// TwinCAT 3 PLC project PLC
// ProgramVersion: 3.1.4023.0
// libraries:
//   Tc2_Standard, * (Beckhoff Automation GmbH)
//   Tc2_System, * (Beckhoff Automation GmbH)
//   Tc3_Module, * (Beckhoff Automation GmbH)
// project tree:
//   / PlcTask.TcTTO
//   POUs/ MAIN.TcPOU
//   DUTs/IO/PdoEntries/ Status_57491DF1.TcDUT, Status_D4FDECD4.TcDUT, Control_0B2F8B70.TcDUT, Status_B0753356.TcDUT, Status_F2CE6D91.TcDUT, Status_3A9E406C.TcDUT, Control_D500AB79.TcDUT, Status_D8D782C3.TcDUT, Control_6EF2C5D0.TcDUT, Status_8CBE219F.TcDUT, Status_B6795845.TcDUT, Control_5FD4673D.TcDUT, Status_1E008DB9.TcDUT, Status_3035BE2E.TcDUT, Control_F189B737.TcDUT, Control_C948E0F2.TcDUT, Status_6CCA259F.TcDUT, Status_72C27E80.TcDUT, Control_254441A5.TcDUT
//   DUTs/IO/PDOs/ InfoData_6F19DB2B.TcDUT, Channel_830843C1.TcDUT, WcState_9091E0EB.TcDUT, Latch_8E413295.TcDUT, WcState_B516A264.TcDUT, InfoData_A7436BC6.TcDUT, CNT_Input_Channel_FF10BD3C.TcDUT, DIG_Inputs_CAFF6004.TcDUT, DIG_Inputs_Device_1F4E72EB.TcDUT, CNT_Output_Channel_550BB6DF.TcDUT, InfoData_32EB74EA.TcDUT, Channel_42CA91F7.TcDUT, WcState_0B2B16F9.TcDUT, Diag_Channel_830843C1.TcDUT, InfoData_0A66F009.TcDUT, AI_Standard_Channel_A8DF64E3.TcDUT, RTD_RTDInputs_Channel_A8DF64E3.TcDUT, AI_Standard_Channel_4A394481.TcDUT, AO_Output_Channel_BA7EBB7C.TcDUT, AI_Inputs_Channel_A8DF64E3.TcDUT, ENC_Status_compact_F4F89583.TcDUT, ENC_Control_compact_E6DC9B25.TcDUT, ENC_Status_compact_7D3464F3.TcDUT, ENC_Control_compact_21E2D14D.TcDUT, COM_Inputs_6C2FC202.TcDUT, COM_Outputs_5D00B5E7.TcDUT, COM_TxPDO_Map_Inputs_Channel_C252EAC2.TcDUT, COM_RxPDO_Map_Outputs_Channel_B336F4EE.TcDUT, COM_TxPDO_Map_Inputs_Channel_6C2FC202.TcDUT, COM_RxPDO_Map_Outputs_Channel_5D00B5E7.TcDUT, ENC_Status_compact_4D066E1A.TcDUT, STM_Status_36ED096F.TcDUT, STM_Control_BA4CE352.TcDUT, STM_Velocity_A47A3F41.TcDUT, InfoData_6538CF5F.TcDUT, STM_Status_DE0D6B37.TcDUT, ENC_Status_compact_Channel_DC559AB0.TcDUT, DCM_Status_Channel_36ED096F.TcDUT, ENC_Control_compact_Channel_2E82BC43.TcDUT, DCM_Control_Channel_5A8B5016.TcDUT, DCM_Velocity_Channel_A47A3F41.TcDUT, InfoData_939F71B6.TcDUT, TACHO_Single_Shaft_Mode_Input_Channel_C331CA3E.TcDUT, DIG_Inputs_495F5DA4.TcDUT, PWM_Status_77939B11.TcDUT, DEV_Inputs_FBF180A4.TcDUT, TACHO_Output_Channel_600697D9.TcDUT, DIG_Outputs_0E284394.TcDUT, PWM_Control_63F162E4.TcDUT, InfoData_E68C61CD.TcDUT, InfoData_2A97D6CF.TcDUT, Inputs_25A0042B.TcDUT, Outputs_2397A10E.TcDUT
//   DUTs/IO/Boxes/ EK1100_1FC0878B.TcDUT, EK1122_1FC0878B.TcDUT, ER1008_78E8D3DD.TcDUT, ER1018_78E8D3DD.TcDUT, ER1098_78E8D3DD.TcDUT, ER1258_58F475DD.TcDUT, ER1518_CC442588.TcDUT, ER1809_32157CFD.TcDUT, ER1819_32157CFD.TcDUT, ER2008_E2806B95.TcDUT, ER2028_E2806B95.TcDUT, ER2038_3AE10DD7.TcDUT, ER2308_F6D9A8D1.TcDUT, ER2318_F6D9A8D1.TcDUT, ER2328_F6D9A8D1.TcDUT, ER2338_7699BCF6.TcDUT, ER2339_D8E9F29A.TcDUT, ER2339_4CF33DED.TcDUT, ER2349_4CF33DED.TcDUT, ER2624_7B64371E.TcDUT, ER2809_2B6483BD.TcDUT, ER3174_DCC78662.TcDUT, ER3184_DCC78662.TcDUT, ER3204_6CD7E119.TcDUT, ER3204_AB25C3AC.TcDUT, ER3314_E65CDB1C.TcDUT, ER4174_AB92710E.TcDUT, ER4374_A304750F.TcDUT, ER5101_87AC78CF.TcDUT, ER5151_7476E948.TcDUT, ER6001_40883D03.TcDUT, ER6002_7F53816A.TcDUT, ER6002_7BE6B617.TcDUT, ER7041_3210CF40.TcDUT, ER7041_3E4BEAEF.TcDUT, ER7342_2AE9C6B3.TcDUT, ER8309_A0C54F77.TcDUT
//   DUTs/IO/Devices/ SyncUnitTask_2D604ED5.TcDUT, SyncUnitTasks_6FEB8257.TcDUT, SyncUnits_99E584AF.TcDUT
//   DUTs/IO/Topology/ Beckhoff_ER1xxxEK1122_4914C526.TcDUT, Beckhoff_ER1xxx_A63E075A.TcDUT, Beckhoff_ER2xxxEK1122_73471FC4.TcDUT, Beckhoff_ER2xxx_CED8BB26.TcDUT, Beckhoff_ER3xxxEK1122_4F8E32D9.TcDUT, Beckhoff_ER3xxx_58A653D9.TcDUT, Beckhoff_ER4xxxEK1122_5C895096.TcDUT, Beckhoff_ER4xxx_797AEBB5.TcDUT, Beckhoff_ER5xxxEK1122_B89AF081.TcDUT, Beckhoff_ER5xxx_22A4CB20.TcDUT, Beckhoff_ER6xxxEK1122_BD5112F1.TcDUT, Beckhoff_ER6xxx_896D799E.TcDUT, Beckhoff_ER7xxxEK1122_0EBE6E72.TcDUT, Beckhoff_ER7xxx_FFC5AE47.TcDUT, Beckhoff_ER8xxxEK1122_CCFAC454.TcDUT, Beckhoff_ER8xxx_509945A9.TcDUT, EtherCAT_Master_ERxxxx_879C9A05.TcDUT
//   DUTs/IO/Base/ EtcSlaveBase_82538BE2.TcDUT, EtcSlaveBase_82538BE2.TcDUT, EtcSlaveBase_82538BE2.TcDUT, EtcSlaveTerminalBase_947E5A46.TcDUT, EtcSlaveBoxBase_77A0E4A7.TcDUT, EtcSlaveEndTerminalBase_866C7F0C.TcDUT, InputBase_8311D824.TcDUT, OutputBase_10CEE7DE.TcDUT, EtcMasterBase_62654B43.TcDUT
//   GVLs/ GVL_iXlinker.TcGVL
// real-time tasks:
//   TASK PlcTask: cycle T#10ms, priority 20, ADS port 350
// I/O:
//   DEVICE EtherCAT_Master_ERxxxx, AmsNetId 172.20.30.238.16.1
//     Beckhoff ER1xxx [EK1100 EtherCAT Coupler (2A E-Bus)]
//       Beckhoff ER1xxxEK1122 [EK1122 2 port EtherCAT junction]
//         Beckhoff ER1xxxsub EK1100 [EK1100 EtherCAT Coupler (2A E-Bus)]
//         A_0001(ER1008-0001-0016) [ER1008-0001 8 Ch. Dig. Input 24V, 3ms, M8]
//         A_0002(ER1008-0001-0018) [ER1008-0001 8 Ch. Dig. Input 24V, 3ms, M8]
//         A_0003(ER1008-0002-0018) [ER1008-0002 8 Ch. Dig. Input 24V, 3ms, M12]
//         A_0004(ER1008-0022-0017) [ER1008-0022 8 Ch. Dig. Input 24V, 3ms, M12]
//         A_0005(ER1018-0001-0018) [ER1018-0001 8 Ch. Dig. Input 24V, 10µs, M8]
//         A_0006(ER1018-0002-0018) [ER1018-0002 8 Ch. Dig. Input 24V, 10µs, M12]
//         A_0007(ER1098-0001-0017) [ER1098-0001 8 Ch. Dig. Input 24V, 10us, M8, negative]
//         A_0008(ER1258-0001-0019) [ER1258-0001 8 Ch. Dig. Input 24V, 10µs, DC Latch, M8]
//         A_0009(ER1258-0001-0020) [ER1258-0001 8 Ch. Dig. Input 24V, 10µs, DC Latch, M8]
//         A_0010(ER1258-0002-0019) [ER1258-0002 8 Ch. Dig. Input 24V, 10µs, DC Latch, M12]
//         A_0011(ER1258-0002-0020) [ER1258-0002 8 Ch. Dig. Input 24V, 10µs, DC Latch, M12]
//         A_0012(ER1518-0002-0018) [ER1518-0002 8 Ch.digital multi-function input]
//         A_0013(ER1518-0002-0019) [ER1518-0002 8 Ch.digital multi-function input]
//         A_0014(ER1809-0021-0017) [ER1809-0021 16 Ch. Dig. Input 24V, 3ms, M8]
//         A_0015(ER1809-0022-0018) [ER1809-0022 16 Ch. Dig. Input 24V, 3ms, M12]
//         A_0016(ER1819-0021-0017) [ER1819-0021 16 Ch. Dig. Input 24V, 10µs, M8]
//         A_0017(ER1819-0022-0017) [ER1819-0022 16 Ch. Dig. Input 24V, 10µs, M12]
//     Beckhoff ER2xxx [EK1100 EtherCAT Coupler (2A E-Bus)]
//       Beckhoff ER2xxxEK1122 [EK1122 2 port EtherCAT junction]
//         Beckhoff ER2xxxsub EK1100 [EK1100 EtherCAT Coupler (2A E-Bus)]
//         A_0001(ER2008-0001-0018) [ER2008-0001 8 Ch. Dig. Output 24V, 0,5A, M8]
//         A_0002(ER2008-0001-0019) [ER2008-0001 8 Ch. Dig. Output 24V, 0,5A, M8]
//         A_0003(ER2008-0002-0018) [ER2008-0002 8 Ch. Dig. Output 24V, 0,5A, M12]
//         A_0004(ER2008-0002-0019) [ER2008-0002 8 Ch. Dig. Output 24V, 0,5A, M12]
//         A_0005(ER2008-0022-0017) [ER2008-0022 8 Ch. Dig. Output 24V, 0,5A, M12]
//         A_0006(ER2008-0022-0018) [ER2008-0022 8 Ch. Dig. Output 24V, 0,5A, M12]
//         A_0007(ER2028-0001-0017) [ER2028-0001 8 Ch. Dig. Output 24V, 2A, M8]
//         A_0008(ER2028-0001-0018) [ER2028-0001 8 Ch. Dig. Output 24V, 2A, M8]
//         A_0009(ER2028-0002-0018) [ER2028-0002 8 Ch. Dig. Output 24V, 2A, M12]
//         A_0010(ER2028-0002-0019) [ER2028-0002 8 Ch. Dig. Output 24V, 2A, M12]
//         A_0011(ER2028-1032-0016) [ER2028-1032 8 Ch. Dig. Output 24V, 2,8A, M12]
//         A_0012(ER2038-0001-0017) [ER2038-0001 8 Ch. Dig. Output 24V, 2A, M8, Diagnostic]
//         A_0013(ER2038-0001-0018) [ER2038-0001 8 Ch. Dig. Output 24V, 2A, M8, Diagnostic]
//         A_0014(ER2038-0002-0017) [ER2038-0002 8 Ch. Dig. Output 24V, 2A, M12, Diagnostic]
//         A_0015(ER2038-0002-0018) [ER2038-0002 8 Ch. Dig. Output 24V, 2A, M12, Diagnostic]
//         A_0016(ER2308-0001-0018) [ER2308-0001 4 Ch. Dig. In, 3ms, 4 Ch. Dig. Out 24V, 0,5A, M8]
//         A_0017(ER2308-0001-0019) [ER2308-0001 4 Ch. Dig. In, 3ms, 4 Ch. Dig. Out 24V, 0,5A, M8]
//         A_0018(ER2308-0002-0018) [ER2308-0002 4 CH. Dig. In, 3ms, 4 Ch. Dig. Out 24V, 0,5A, M12]
//         A_0019(ER2308-0002-0019) [ER2308-0002 4 CH. Dig. In, 3ms, 4 Ch. Dig. Out 24V, 0,5A, M12]
//         A_0020(ER2318-0001-0018) [ER2318-0001 4 Ch. Dig. In, 10µs, 4 Ch. Dig. Out 24V, 0,5A, M8]
//         A_0021(ER2318-0001-0019) [ER2318-0001 4 Ch. Dig. In, 10µs, 4 Ch. Dig. Out 24V, 0,5A, M8]
//         A_0022(ER2318-0002-0018) [ER2318-0002 4 Ch. Dig. In, 10µs, 4 Ch. Dig. Out 24V, 0,5A, M12]
//         A_0023(ER2318-0002-0019) [ER2318-0002 4 Ch. Dig. In, 10µs, 4 Ch. Dig. Out 24V, 0,5A, M12]
//         A_0024(ER2328-0001-0017) [ER2328-0001 4 CH. Dig. In, 3ms, 4 Ch. Dig. Out 24V, 2A, M8]
//         A_0025(ER2328-0001-0018) [ER2328-0001 4 CH. Dig. In, 3ms, 4 Ch. Dig. Out 24V, 2A, M8]
//         A_0026(ER2328-0002-0018) [ER2328-0002 4 CH. Dig. In, 3ms, 4 Ch. Dig. Out 24V, 2A, M12]
//         A_0027(ER2328-0002-0019) [ER2328-0002 4 CH. Dig. In, 3ms, 4 Ch. Dig. Out 24V, 2A, M12]
//         A_0028(ER2338-0001-0022) [ER2338-0001 8 Ch. Dig. Input/Output 24V, 0,5A, M8]
//         A_0029(ER2338-0001-0023) [ER2338-0001 8 Ch. Dig. Input/Output 24V, 0,5A, M8]
//         A_0030(ER2338-0002-0022) [ER2338-0002 8 Ch. Dig. Input/Output 24V, 0,5A, M12]
//         A_0031(ER2338-0002-0023) [ER2338-0002 8 Ch. Dig. Input/Output 24V, 0,5A, M12]
//         A_0032(ER2338-1001-0017) [ER2338-1001 8 Ch. Dig. Input/Output 24V, 3ms, 0,5A, M8]
//         A_0033(ER2338-1001-0018) [ER2338-1001 8 Ch. Dig. Input/Output 24V, 3ms, 0,5A, M8]
//         A_0034(ER2338-1002-0017) [ER2338-1002 8 Ch. Dig. Input/Output 24V, 3ms, 0,5A, M12]
//         A_0035(ER2338-1002-0018) [ER2338-1002 8 Ch. Dig. Input/Output 24V, 3ms, 0,5A, M12]
//         A_0036(ER2339-0021-0018) [ER2339-0021 16 Ch. Dig. Input/Output 24V, 0,5A, M8]
//         A_0037(ER2339-0021-0019) [ER2339-0021 16 Ch. Dig. Input/Output 24V, 0,5A, M8]
//         A_0038(ER2339-0022-0018) [ER2339-0022 16 Ch. Dig. Input/Output 24V, 0,5A, M12]
//         A_0039(ER2339-0022-0019) [ER2339-0022 16 Ch. Dig. Input/Output 24V, 0,5A, M12]
//         A_0040(ER2349-0021-0017) [ER2349-0021 16 Ch. Dig. Input/Output 24V, 10µs, 0,5A, M8]
//         A_0041(ER2349-0021-0018) [ER2349-0021 16 Ch. Dig. Input/Output 24V, 10µs, 0,5A, M8]
//         A_0042(ER2349-0022-0017) [ER2349-0022 16 Ch. Dig. Input/Output 24V, 10µs, 0,5A, M12]
//         A_0043(ER2349-0022-0018) [ER2349-0022 16 Ch. Dig. Input/Output 24V, 10µs, 0,5A, M12]
//         A_0044(ER2624-0002-0018) [ER2624-0002 4Ch. Relay Output, NO (125V AC / 30V DC)]
//         A_0045(ER2624-0002-0019) [ER2624-0002 4Ch. Relay Output, NO (125V AC / 30V DC)]
//         A_0046(ER2809-0021-0017) [ER2809-0021 16 Ch. Dig. Output 24V, 0,5A, M8]
//         A_0047(ER2809-0021-0018) [ER2809-0021 16 Ch. Dig. Output 24V, 0,5A, M8]
//         A_0048(ER2809-0022-0016) [ER2809-0022 16 Ch. Dig. Output 24V, 0,5A, M12]
//         A_0049(ER2809-0022-0017) [ER2809-0022 16 Ch. Dig. Output 24V, 0,5A, M12]
//         A_0050(ER2809-0022-0018) [ER2809-0022 16 Ch. Dig. Output 24V, 0,5A, M12]
//     Beckhoff ER3xxx [EK1100 EtherCAT Coupler (2A E-Bus)]
//       Beckhoff ER3xxxEK1122 [EK1122 2 port EtherCAT junction]
//         Beckhoff ER3xxxsub EK1100 [EK1100 EtherCAT Coupler (2A E-Bus)]
//         A_0001(ER3174-0002-0016) [ER3174-0002 4Ch. Ana. Input +/-10V, 0-10V, 0/4-20mA configurable]
//         A_0002(ER3174-0002-0022) [ER3174-0002 4Ch. Ana. Input +/-10V, 0-10V, 0/4-20mA configurable]
//         A_0003(ER3174-0002-0023) [ER3174-0002 4Ch. Ana. Input +/-10V, 0-10V, 0/4-20mA configurable]
//         A_0004(ER3184-0002-0019) [ER3184-0002 4Ch. Ana. Input +/-10V, 0-10V, 0/4-20mA configurable, single ended]
//         A_0005(ER3184-0002-0020) [ER3184-0002 4Ch. Ana. Input +/-10V, 0-10V, 0/4-20mA configurable, single ended]
//         A_0006(ER3184-0002-0021) [ER3184-0002 4Ch. Ana. Input +/-10V, 0-10V, 0/4-20mA configurable, single ended]
//         A_0007(ER3184-1002-0020) [ER3184-1002 4Ch. Ana. Input +/-10V, 0-10V, 0/4-20mA configurable, single ended]
//         A_0008(ER3184-1002-0021) [ER3184-1002 4Ch. Ana. Input +/-10V, 0-10V, 0/4-20mA configurable, single ended]
//         A_0009(ER3204-0002-0016) [ER3204-0002 4Ch. Ana. Input PT100 (RTD)]
//         A_0010(ER3204-0002-0020) [ER3204-0002 4Ch. Ana. Input PT100 (RTD)]
//         A_0011(ER3204-0002-0021) [ER3204-0002 4Ch. Ana. Input PT100 (RTD)]
//         A_0012(ER3314-0002-0021) [ER3314-0002 4Ch. Ana. Input Thermocouple (TC)]
//     Beckhoff ER4xxx [EK1100 EtherCAT Coupler (2A E-Bus)]
//       Beckhoff ER4xxxEK1122 [EK1122 2 port EtherCAT junction]
//         Beckhoff ER4xxxsub EK1100 [EK1100 EtherCAT Coupler (2A E-Bus)]
//         A_0001(ER4174-0002-0016) [ER4174-0002 4Ch. Ana. Output +/-10V, 0-10V, 0/4-20mA configurable]
//         A_0002(ER4174-0002-0019) [ER4174-0002 4Ch. Ana. Output +/-10V, 0-10V, 0/4-20mA configurable]
//         A_0003(ER4374-0002-0018) [ER4374-0002 2Ch. Ana. Input +/-10V, 0-10V, 0/4-20mA configurable; 2Ch. Ana. Output +/-10V, 0-10V, 0/4-20mA configurable]
//         A_0004(ER4374-0002-0019) [ER4374-0002 2Ch. Ana. Input +/-10V, 0-10V, 0/4-20mA configurable; 2Ch. Ana. Output +/-10V, 0-10V, 0/4-20mA configurable]
//     Beckhoff ER5xxx [EK1100 EtherCAT Coupler (2A E-Bus)]
//       Beckhoff ER5xxxEK1122 [EK1122 2 port EtherCAT junction]
//         Beckhoff ER5xxxsub EK1100 [EK1100 EtherCAT Coupler (2A E-Bus)]
//         A_0001(ER5101-0002-0019) [ER5101-0002 1Ch. Inc. Encoder 5V, M12]
//         A_0002(ER5101-1002-0017) [ER5101-1002 1Ch. Inc. Encoder 5V, M12, 24V Sensor Supply]
//         A_0003(ER5151-0002-0018) [ER5151-0002 1Ch. Inc. Encoder 24V, M12, single ended]
//     Beckhoff ER6xxx [EK1100 EtherCAT Coupler (2A E-Bus)]
//       Beckhoff ER6xxxEK1122 [EK1122 2 port EtherCAT junction]
//         Beckhoff ER6xxxsub EK1100 [EK1100 EtherCAT Coupler (2A E-Bus)]
//         A_0001(ER6001-0002-0016) [ER6001-0002 Interface (RS232/422/485)]
//         A_0002(ER6001-0002-0021) [ER6001-0002 Interface (RS232/422/485)]
//         A_0003(ER6002-0002-0021) [ER6002-0002 Interface (RS232/422/485)]
//         A_0004(ER6002-0002-0022) [ER6002-0002 Interface (RS232/422/485)]
//         A_0005(ER6002-0002-0023) [ER6002-0002 Interface (RS232/422/485)]
//     Beckhoff ER7xxx [EK1100 EtherCAT Coupler (2A E-Bus)]
//       Beckhoff ER7xxxEK1122 [EK1122 2 port EtherCAT junction]
//         Beckhoff ER7xxxsub EK1100 [EK1100 EtherCAT Coupler (2A E-Bus)]
//         A_0001(ER7041-0002-0024) [ER7041-0002 1Ch. Stepper motor output stage (50V, 5A)]
//         A_0002(ER7041-0002-0025) [ER7041-0002 1Ch. Stepper motor output stage (50V, 5A)]
//         A_0003(ER7041-1002-0024) [ER7041-1002 1Ch. Stepper motor output stage (50V, 1.5A)]
//         A_0004(ER7041-1002-0025) [ER7041-1002 1Ch. Stepper motor output stage (50V, 1.5A)]
//         A_0005(ER7041-2002-0024) [ER7041-2002 1Ch. Stepper motor output stage (50V, 5A)]
//         A_0006(ER7041-2002-0025) [ER7041-2002 1Ch. Stepper motor output stage (50V, 5A)]
//         A_0007(ER7041-3002-0021) [ER7041-3002 1Ch. Stepper motor output stage (50V, 5A)]
//         A_0008(ER7041-3002-0022) [ER7041-3002 1Ch. Stepper motor output stage (50V, 5A)]
//         A_0009(ER7342-0002-0020) [ER7342-0002 2Ch. DC motor output stage (50V, 3.5A)]
//         A_0010(ER7342-0002-0021) [ER7342-0002 2Ch. DC motor output stage (50V, 3.5A)]
//         A_0011(ER7342-0002-0022) [ER7342-0002 2Ch. DC motor output stage (50V, 3.5A)]
//     Beckhoff ER8xxx [EK1100 EtherCAT Coupler (2A E-Bus)]
//       Beckhoff ER8xxxEK1122 [EK1122 2 port EtherCAT junction]
//         Beckhoff ER8xxxsub EK1100 [EK1100 EtherCAT Coupler (2A E-Bus)]
//         A_0001(ER8309-1022-0018) [ER8309-1022 2Ch. Ana. Input 4-20mA, 1Ch. Pulse Width Current Output (24V, 1.2A), 1 Ch Ana. Output, 2Ch Dig. Out 24V, 0.5A, 4Ch Dig. In. 24V, 4Ch Dig In/Out 24V, 0.5A, M12]
// variable links:
//   PLC/PLC Instance <-> EtherCAT Master ERxxxx/Beckhoff ER1xxx
//     PlcTask Inputs/GVL_iXlinker.EtherCAT_Master_ERxxxx.Beckhoff_ER1xxx.InfoData.State <-> InfoData/State
//   PLC/PLC Instance <-> EtherCAT Master ERxxxx/Beckhoff ER1xxx/Beckhoff ER1xxxEK1122
//     PlcTask Inputs/GVL_iXlinker.EtherCAT_Master_ERxxxx.Beckhoff_ER1xxx.Beckhoff_ER1xxxEK1122.InfoData.State <-> InfoData/State
//   PLC/PLC Instance <-> EtherCAT Master ERxxxx/Beckhoff ER1xxx/Beckhoff ER1xxxEK1122/Beckhoff ER1xxxsub EK1100
//     PlcTask Inputs/GVL_iXlinker.EtherCAT_Master_ERxxxx.Beckhoff_ER1xxx.Beckhoff_ER1xxxEK1122.Beckhoff_ER1xxxsub_EK1100.InfoData.State <-> InfoData/State
//   PLC/PLC Instance <-> EtherCAT Master ERxxxx/Beckhoff ER1xxx/Beckhoff ER1xxxEK1122/A_0001(ER1008-0001-0016)
//     PlcTask Inputs/GVL_iXlinker.EtherCAT_Master_ERxxxx.Beckhoff_ER1xxx.Beckhoff_ER1xxxEK1122.A_0001_ER1008_0001_0016.Channel_1.Input <-> Channel 1/Input
//     PlcTask Inputs/GVL_iXlinker.EtherCAT_Master_ERxxxx.Beckhoff_ER1xxx.Beckhoff_ER1xxxEK1122.A_0001_ER1008_0001_0016.Channel_2.Input <-> Channel 2/Input
//     PlcTask Inputs/GVL_iXlinker.EtherCAT_Master_ERxxxx.Beckhoff_ER1xxx.Beckhoff_ER1xxxEK1122.A_0001_ER1008_0001_0016.Channel_3.Input <-> Channel 3/Input
//     PlcTask Inputs/GVL_iXlinker.EtherCAT_Master_ERxxxx.Beckhoff_ER1xxx.Beckhoff_ER1xxxEK1122.A_0001_ER1008_0001_0016.Channel_4.Input <-> Channel 4/Input
//     PlcTask Inputs/GVL_iXlinker.EtherCAT_Master_ERxxxx.Beckhoff_ER1xxx.Beckhoff_ER1xxxEK1122.A_0001_ER1008_0001_0016.Channel_5.Input <-> Channel 5/Input
//     PlcTask Inputs/GVL_iXlinker.EtherCAT_Master_ERxxxx.Beckhoff_ER1xxx.Beckhoff_ER1xxxEK1122.A_0001_ER1008_0001_0016.Channel_6.Input <-> Channel 6/Input
//     PlcTask Inputs/GVL_iXlinker.EtherCAT_Master_ERxxxx.Beckhoff_ER1xxx.Beckhoff_ER1xxxEK1122.A_0001_ER1008_0001_0016.Channel_7.Input <-> Channel 7/Input
//     PlcTask Inputs/GVL_iXlinker.EtherCAT_Master_ERxxxx.Beckhoff_ER1xxx.Beckhoff_ER1xxxEK1122.A_0001_ER1008_0001_0016.Channel_8.Input <-> Channel 8/Input
//     PlcTask Inputs/GVL_iXlinker.EtherCAT_Master_ERxxxx.Beckhoff_ER1xxx.Beckhoff_ER1xxxEK1122.A_0001_ER1008_0001_0016.WcState.WcState <-> WcState/WcState
//     PlcTask Inputs/GVL_iXlinker.EtherCAT_Master_ERxxxx.Beckhoff_ER1xxx.Beckhoff_ER1xxxEK1122.A_0001_ER1008_0001_0016.WcState.InputToggle <-> WcState/InputToggle
//     PlcTask Inputs/GVL_iXlinker.EtherCAT_Master_ERxxxx.Beckhoff_ER1xxx.Beckhoff_ER1xxxEK1122.A_0001_ER1008_0001_0016.InfoData.State <-> InfoData/State
//   PLC/PLC Instance <-> EtherCAT Master ERxxxx/Beckhoff ER1xxx/Beckhoff ER1xxxEK1122/A_0002(ER1008-0001-0018)
//     PlcTask Inputs/GVL_iXlinker.EtherCAT_Master_ERxxxx.Beckhoff_ER1xxx.Beckhoff_ER1xxxEK1122.A_0002_ER1008_0001_0018.Channel_1.Input <-> Channel 1/Input
//     PlcTask Inputs/GVL_iXlinker.EtherCAT_Master_ERxxxx.Beckhoff_ER1xxx.Beckhoff_ER1xxxEK1122.A_0002_ER1008_0001_0018.Channel_2.Input <-> Channel 2/Input
//     PlcTask Inputs/GVL_iXlinker.EtherCAT_Master_ERxxxx.Beckhoff_ER1xxx.Beckhoff_ER1xxxEK1122.A_0002_ER1008_0001_0018.Channel_3.Input <-> Channel 3/Input
//     PlcTask Inputs/GVL_iXlinker.EtherCAT_Master_ERxxxx.Beckhoff_ER1xxx.Beckhoff_ER1xxxEK1122.A_0002_ER1008_0001_0018.Channel_4.Input <-> Channel 4/Input
//     PlcTask Inputs/GVL_iXlinker.EtherCAT_Master_ERxxxx.Beckhoff_ER1xxx.Beckhoff_ER1xxxEK1122.A_0002_ER1008_0001_0018.Channel_5.Input <-> Channel 5/Input
//     PlcTask Inputs/GVL_iXlinker.EtherCAT_Master_ERxxxx.Beckhoff_ER1xxx.Beckhoff_ER1xxxEK1122.A_0002_ER1008_0001_0018.Channel_6.Input <-> Channel 6/Input
//     PlcTask Inputs/GVL_iXlinker.EtherCAT_Master_ERxxxx.Beckhoff_ER1xxx.Beckhoff_ER1xxxEK1122.A_0002_ER1008_0001_0018.Channel_7.Input <-> Channel 7/Input
//     PlcTask Inputs/GVL_iXlinker.EtherCAT_Master_ERxxxx.Beckhoff_ER1xxx.Beckhoff_ER1xxxEK1122.A_0002_ER1008_0001_0018.Channel_8.Input <-> Channel 8/Input
//     PlcTask Inputs/GVL_iXlinker.EtherCAT_Master_ERxxxx.Beckhoff_ER1xxx.Beckhoff_ER1xxxEK1122.A_0002_ER1008_0001_0018.WcState.WcState <-> WcState/WcState
//     PlcTask Inputs/GVL_iXlinker.EtherCAT_Master_ERxxxx.Beckhoff_ER1xxx.Beckhoff_ER1xxxEK1122.A_0002_ER1008_0001_0018.WcState.InputToggle <-> WcState/InputToggle
//     PlcTask Inputs/GVL_iXlinker.EtherCAT_Master_ERxxxx.Beckhoff_ER1xxx.Beckhoff_ER1xxxEK1122.A_0002_ER1008_0001_0018.InfoData.State <-> InfoData/State
//   PLC/PLC Instance <-> EtherCAT Master ERxxxx/Beckhoff ER1xxx/Beckhoff ER1xxxEK1122/A_0003(ER1008-0002-0018)
//     PlcTask Inputs/GVL_iXlinker.EtherCAT_Master_ERxxxx.Beckhoff_ER1xxx.Beckhoff_ER1xxxEK1122.A_0003_ER1008_0002_0018.Channel_1.Input <-> Channel 1/Input
//     PlcTask Inputs/GVL_iXlinker.EtherCAT_Master_ERxxxx.Beckhoff_ER1xxx.Beckhoff_ER1xxxEK1122.A_0003_ER1008_0002_0018.Channel_2.Input <-> Channel 2/Input
//     PlcTask Inputs/GVL_iXlinker.EtherCAT_Master_ERxxxx.Beckhoff_ER1xxx.Beckhoff_ER1xxxEK1122.A_0003_ER1008_0002_0018.Channel_3.Input <-> Channel 3/Input
//     PlcTask Inputs/GVL_iXlinker.EtherCAT_Master_ERxxxx.Beckhoff_ER1xxx.Beckhoff_ER1xxxEK1122.A_0003_ER1008_0002_0018.Channel_4.Input <-> Channel 4/Input
//     PlcTask Inputs/GVL_iXlinker.EtherCAT_Master_ERxxxx.Beckhoff_ER1xxx.Beckhoff_ER1xxxEK1122.A_0003_ER1008_0002_0018.Channel_5.Input <-> Channel 5/Input
//     PlcTask Inputs/GVL_iXlinker.EtherCAT_Master_ERxxxx.Beckhoff_ER1xxx.Beckhoff_ER1xxxEK1122.A_0003_ER1008_0002_0018.Channel_6.Input <-> Channel 6/Input
//     PlcTask Inputs/GVL_iXlinker.EtherCAT_Master_ERxxxx.Beckhoff_ER1xxx.Beckhoff_ER1xxxEK1122.A_0003_ER1008_0002_0018.Channel_7.Input <-> Channel 7/Input
//     PlcTask Inputs/GVL_iXlinker.EtherCAT_Master_ERxxxx.Beckhoff_ER1xxx.Beckhoff_ER1xxxEK1122.A_0003_ER1008_0002_0018.Channel_8.Input <-> Channel 8/Input
//     PlcTask Inputs/GVL_iXlinker.EtherCAT_Master_ERxxxx.Beckhoff_ER1xxx.Beckhoff_ER1xxxEK1122.A_0003_ER1008_0002_0018.WcState.WcState <-> WcState/WcState
//     PlcTask Inputs/GVL_iXlinker.EtherCAT_Master_ERxxxx.Beckhoff_ER1xxx.Beckhoff_ER1xxxEK1122.A_0003_ER1008_0002_0018.WcState.InputToggle <-> WcState/InputToggle
//     PlcTask Inputs/GVL_iXlinker.EtherCAT_Master_ERxxxx.Beckhoff_ER1xxx.Beckhoff_ER1xxxEK1122.A_0003_ER1008_0002_0018.InfoData.State <-> InfoData/State
//   PLC/PLC Instance <-> EtherCAT Master ERxxxx/Beckhoff ER1xxx/Beckhoff ER1xxxEK1122/A_0004(ER1008-0022-0017)
//     PlcTask Inputs/GVL_iXlinker.EtherCAT_Master_ERxxxx.Beckhoff_ER1xxx.Beckhoff_ER1xxxEK1122.A_0004_ER1008_0022_0017.Channel_1.Input <-> Channel 1/Input
//     PlcTask Inputs/GVL_iXlinker.EtherCAT_Master_ERxxxx.Beckhoff_ER1xxx.Beckhoff_ER1xxxEK1122.A_0004_ER1008_0022_0017.Channel_2.Input <-> Channel 2/Input
//     PlcTask Inputs/GVL_iXlinker.EtherCAT_Master_ERxxxx.Beckhoff_ER1xxx.Beckhoff_ER1xxxEK1122.A_0004_ER1008_0022_0017.Channel_3.Input <-> Channel 3/Input
//     PlcTask Inputs/GVL_iXlinker.EtherCAT_Master_ERxxxx.Beckhoff_ER1xxx.Beckhoff_ER1xxxEK1122.A_0004_ER1008_0022_0017.Channel_4.Input <-> Channel 4/Input
//     PlcTask Inputs/GVL_iXlinker.EtherCAT_Master_ERxxxx.Beckhoff_ER1xxx.Beckhoff_ER1xxxEK1122.A_0004_ER1008_0022_0017.Channel_5.Input <-> Channel 5/Input
//     PlcTask Inputs/GVL_iXlinker.EtherCAT_Master_ERxxxx.Beckhoff_ER1xxx.Beckhoff_ER1xxxEK1122.A_0004_ER1008_0022_0017.Channel_6.Input <-> Channel 6/Input
//     PlcTask Inputs/GVL_iXlinker.EtherCAT_Master_ERxxxx.Beckhoff_ER1xxx.Beckhoff_ER1xxxEK1122.A_0004_ER1008_0022_0017.Channel_7.Input <-> Channel 7/Input
//     PlcTask Inputs/GVL_iXlinker.EtherCAT_Master_ERxxxx.Beckhoff_ER1xxx.Beckhoff_ER1xxxEK1122.A_0004_ER1008_0022_0017.Channel_8.Input <-> Channel 8/Input
//     PlcTask Inputs/GVL_iXlinker.EtherCAT_Master_ERxxxx.Beckhoff_ER1xxx.Beckhoff_ER1xxxEK1122.A_0004_ER1008_0022_0017.WcState.WcState <-> WcState/WcState
//     PlcTask Inputs/GVL_iXlinker.EtherCAT_Master_ERxxxx.Beckhoff_ER1xxx.Beckhoff_ER1xxxEK1122.A_0004_ER1008_0022_0017.WcState.InputToggle <-> WcState/InputToggle
//     PlcTask Inputs/GVL_iXlinker.EtherCAT_Master_ERxxxx.Beckhoff_ER1xxx.Beckhoff_ER1xxxEK1122.A_0004_ER1008_0022_0017.InfoData.State <-> InfoData/State
//   PLC/PLC Instance <-> EtherCAT Master ERxxxx/Beckhoff ER1xxx/Beckhoff ER1xxxEK1122/A_0005(ER1018-0001-0018)
//     PlcTask Inputs/GVL_iXlinker.EtherCAT_Master_ERxxxx.Beckhoff_ER1xxx.Beckhoff_ER1xxxEK1122.A_0005_ER1018_0001_0018.Channel_1.Input <-> Channel 1/Input
//     PlcTask Inputs/GVL_iXlinker.EtherCAT_Master_ERxxxx.Beckhoff_ER1xxx.Beckhoff_ER1xxxEK1122.A_0005_ER1018_0001_0018.Channel_2.Input <-> Channel 2/Input
//     PlcTask Inputs/GVL_iXlinker.EtherCAT_Master_ERxxxx.Beckhoff_ER1xxx.Beckhoff_ER1xxxEK1122.A_0005_ER1018_0001_0018.Channel_3.Input <-> Channel 3/Input
//     PlcTask Inputs/GVL_iXlinker.EtherCAT_Master_ERxxxx.Beckhoff_ER1xxx.Beckhoff_ER1xxxEK1122.A_0005_ER1018_0001_0018.Channel_4.Input <-> Channel 4/Input
//     PlcTask Inputs/GVL_iXlinker.EtherCAT_Master_ERxxxx.Beckhoff_ER1xxx.Beckhoff_ER1xxxEK1122.A_0005_ER1018_0001_0018.Channel_5.Input <-> Channel 5/Input
//     PlcTask Inputs/GVL_iXlinker.EtherCAT_Master_ERxxxx.Beckhoff_ER1xxx.Beckhoff_ER1xxxEK1122.A_0005_ER1018_0001_0018.Channel_6.Input <-> Channel 6/Input
//     PlcTask Inputs/GVL_iXlinker.EtherCAT_Master_ERxxxx.Beckhoff_ER1xxx.Beckhoff_ER1xxxEK1122.A_0005_ER1018_0001_0018.Channel_7.Input <-> Channel 7/Input
//     PlcTask Inputs/GVL_iXlinker.EtherCAT_Master_ERxxxx.Beckhoff_ER1xxx.Beckhoff_ER1xxxEK1122.A_0005_ER1018_0001_0018.Channel_8.Input <-> Channel 8/Input
//     PlcTask Inputs/GVL_iXlinker.EtherCAT_Master_ERxxxx.Beckhoff_ER1xxx.Beckhoff_ER1xxxEK1122.A_0005_ER1018_0001_0018.WcState.WcState <-> WcState/WcState
//     PlcTask Inputs/GVL_iXlinker.EtherCAT_Master_ERxxxx.Beckhoff_ER1xxx.Beckhoff_ER1xxxEK1122.A_0005_ER1018_0001_0018.WcState.InputToggle <-> WcState/InputToggle
//     PlcTask Inputs/GVL_iXlinker.EtherCAT_Master_ERxxxx.Beckhoff_ER1xxx.Beckhoff_ER1xxxEK1122.A_0005_ER1018_0001_0018.InfoData.State <-> InfoData/State
//   PLC/PLC Instance <-> EtherCAT Master ERxxxx/Beckhoff ER1xxx/Beckhoff ER1xxxEK1122/A_0006(ER1018-0002-0018)
//     PlcTask Inputs/GVL_iXlinker.EtherCAT_Master_ERxxxx.Beckhoff_ER1xxx.Beckhoff_ER1xxxEK1122.A_0006_ER1018_0002_0018.Channel_1.Input <-> Channel 1/Input
//     PlcTask Inputs/GVL_iXlinker.EtherCAT_Master_ERxxxx.Beckhoff_ER1xxx.Beckhoff_ER1xxxEK1122.A_0006_ER1018_0002_0018.Channel_2.Input <-> Channel 2/Input
//     PlcTask Inputs/GVL_iXlinker.EtherCAT_Master_ERxxxx.Beckhoff_ER1xxx.Beckhoff_ER1xxxEK1122.A_0006_ER1018_0002_0018.Channel_3.Input <-> Channel 3/Input
//     PlcTask Inputs/GVL_iXlinker.EtherCAT_Master_ERxxxx.Beckhoff_ER1xxx.Beckhoff_ER1xxxEK1122.A_0006_ER1018_0002_0018.Channel_4.Input <-> Channel 4/Input
//     PlcTask Inputs/GVL_iXlinker.EtherCAT_Master_ERxxxx.Beckhoff_ER1xxx.Beckhoff_ER1xxxEK1122.A_0006_ER1018_0002_0018.Channel_5.Input <-> Channel 5/Input
//     PlcTask Inputs/GVL_iXlinker.EtherCAT_Master_ERxxxx.Beckhoff_ER1xxx.Beckhoff_ER1xxxEK1122.A_0006_ER1018_0002_0018.Channel_6.Input <-> Channel 6/Input
//     PlcTask Inputs/GVL_iXlinker.EtherCAT_Master_ERxxxx.Beckhoff_ER1xxx.Beckhoff_ER1xxxEK1122.A_0006_ER1018_0002_0018.Channel_7.Input <-> Channel 7/Input
//     PlcTask Inputs/GVL_iXlinker.EtherCAT_Master_ERxxxx.Beckhoff_ER1xxx.Beckhoff_ER1xxxEK1122.A_0006_ER1018_0002_0018.Channel_8.Input <-> Channel 8/Input
//     PlcTask Inputs/GVL_iXlinker.EtherCAT_Master_ERxxxx.Beckhoff_ER1xxx.Beckhoff_ER1xxxEK1122.A_0006_ER1018_0002_0018.WcState.WcState <-> WcState/WcState
//     PlcTask Inputs/GVL_iXlinker.EtherCAT_Master_ERxxxx.Beckhoff_ER1xxx.Beckhoff_ER1xxxEK1122.A_0006_ER1018_0002_0018.WcState.InputToggle <-> WcState/InputToggle
//     PlcTask Inputs/GVL_iXlinker.EtherCAT_Master_ERxxxx.Beckhoff_ER1xxx.Beckhoff_ER1xxxEK1122.A_0006_ER1018_0002_0018.InfoData.State <-> InfoData/State
//   PLC/PLC Instance <-> EtherCAT Master ERxxxx/Beckhoff ER1xxx/Beckhoff ER1xxxEK1122/A_0007(ER1098-0001-0017)
//     PlcTask Inputs/GVL_iXlinker.EtherCAT_Master_ERxxxx.Beckhoff_ER1xxx.Beckhoff_ER1xxxEK1122.A_0007_ER1098_0001_0017.Channel_1.Input <-> Channel 1/Input
//     PlcTask Inputs/GVL_iXlinker.EtherCAT_Master_ERxxxx.Beckhoff_ER1xxx.Beckhoff_ER1xxxEK1122.A_0007_ER1098_0001_0017.Channel_2.Input <-> Channel 2/Input
//     PlcTask Inputs/GVL_iXlinker.EtherCAT_Master_ERxxxx.Beckhoff_ER1xxx.Beckhoff_ER1xxxEK1122.A_0007_ER1098_0001_0017.Channel_3.Input <-> Channel 3/Input
//     PlcTask Inputs/GVL_iXlinker.EtherCAT_Master_ERxxxx.Beckhoff_ER1xxx.Beckhoff_ER1xxxEK1122.A_0007_ER1098_0001_0017.Channel_4.Input <-> Channel 4/Input
//     PlcTask Inputs/GVL_iXlinker.EtherCAT_Master_ERxxxx.Beckhoff_ER1xxx.Beckhoff_ER1xxxEK1122.A_0007_ER1098_0001_0017.Channel_5.Input <-> Channel 5/Input
//     PlcTask Inputs/GVL_iXlinker.EtherCAT_Master_ERxxxx.Beckhoff_ER1xxx.Beckhoff_ER1xxxEK1122.A_0007_ER1098_0001_0017.Channel_6.Input <-> Channel 6/Input
//     PlcTask Inputs/GVL_iXlinker.EtherCAT_Master_ERxxxx.Beckhoff_ER1xxx.Beckhoff_ER1xxxEK1122.A_0007_ER1098_0001_0017.Channel_7.Input <-> Channel 7/Input
//     PlcTask Inputs/GVL_iXlinker.EtherCAT_Master_ERxxxx.Beckhoff_ER1xxx.Beckhoff_ER1xxxEK1122.A_0007_ER1098_0001_0017.Channel_8.Input <-> Channel 8/Input
//     PlcTask Inputs/GVL_iXlinker.EtherCAT_Master_ERxxxx.Beckhoff_ER1xxx.Beckhoff_ER1xxxEK1122.A_0007_ER1098_0001_0017.WcState.WcState <-> WcState/WcState
//     PlcTask Inputs/GVL_iXlinker.EtherCAT_Master_ERxxxx.Beckhoff_ER1xxx.Beckhoff_ER1xxxEK1122.A_0007_ER1098_0001_0017.WcState.InputToggle <-> WcState/InputToggle
//     PlcTask Inputs/GVL_iXlinker.EtherCAT_Master_ERxxxx.Beckhoff_ER1xxx.Beckhoff_ER1xxxEK1122.A_0007_ER1098_0001_0017.InfoData.State <-> InfoData/State
//   PLC/PLC Instance <-> EtherCAT Master ERxxxx/Beckhoff ER1xxx/Beckhoff ER1xxxEK1122/A_0008(ER1258-0001-0019)
//     PlcTask Inputs/GVL_iXlinker.EtherCAT_Master_ERxxxx.Beckhoff_ER1xxx.Beckhoff_ER1xxxEK1122.A_0008_ER1258_0001_0019.Channel_1.Input <-> Channel 1/Input
//     PlcTask Inputs/GVL_iXlinker.EtherCAT_Master_ERxxxx.Beckhoff_ER1xxx.Beckhoff_ER1xxxEK1122.A_0008_ER1258_0001_0019.Channel_2.Input <-> Channel 2/Input
//     PlcTask Inputs/GVL_iXlinker.EtherCAT_Master_ERxxxx.Beckhoff_ER1xxx.Beckhoff_ER1xxxEK1122.A_0008_ER1258_0001_0019.Channel_3.Input <-> Channel 3/Input
//     PlcTask Inputs/GVL_iXlinker.EtherCAT_Master_ERxxxx.Beckhoff_ER1xxx.Beckhoff_ER1xxxEK1122.A_0008_ER1258_0001_0019.Channel_4.Input <-> Channel 4/Input
//     PlcTask Inputs/GVL_iXlinker.EtherCAT_Master_ERxxxx.Beckhoff_ER1xxx.Beckhoff_ER1xxxEK1122.A_0008_ER1258_0001_0019.Channel_5.Input <-> Channel 5/Input
//     PlcTask Inputs/GVL_iXlinker.EtherCAT_Master_ERxxxx.Beckhoff_ER1xxx.Beckhoff_ER1xxxEK1122.A_0008_ER1258_0001_0019.Channel_6.Input <-> Channel 6/Input
//     PlcTask Inputs/GVL_iXlinker.EtherCAT_Master_ERxxxx.Beckhoff_ER1xxx.Beckhoff_ER1xxxEK1122.A_0008_ER1258_0001_0019.Channel_7.Input <-> Channel 7/Input
//     PlcTask Inputs/GVL_iXlinker.EtherCAT_Master_ERxxxx.Beckhoff_ER1xxx.Beckhoff_ER1xxxEK1122.A_0008_ER1258_0001_0019.Channel_8.Input <-> Channel 8/Input
//     PlcTask Inputs/GVL_iXlinker.EtherCAT_Master_ERxxxx.Beckhoff_ER1xxx.Beckhoff_ER1xxxEK1122.A_0008_ER1258_0001_0019.Latch.Status0 <-> Latch/Status0
//     PlcTask Inputs/GVL_iXlinker.EtherCAT_Master_ERxxxx.Beckhoff_ER1xxx.Beckhoff_ER1xxxEK1122.A_0008_ER1258_0001_0019.Latch.Status1 <-> Latch/Status1
//     PlcTask Inputs/GVL_iXlinker.EtherCAT_Master_ERxxxx.Beckhoff_ER1xxx.Beckhoff_ER1xxxEK1122.A_0008_ER1258_0001_0019.Latch.LatchPos0 <-> Latch/LatchPos0
//     PlcTask Inputs/GVL_iXlinker.EtherCAT_Master_ERxxxx.Beckhoff_ER1xxx.Beckhoff_ER1xxxEK1122.A_0008_ER1258_0001_0019.Latch.LatchPos1 <-> Latch/LatchPos1
//     PlcTask Inputs/GVL_iXlinker.EtherCAT_Master_ERxxxx.Beckhoff_ER1xxx.Beckhoff_ER1xxxEK1122.A_0008_ER1258_0001_0019.Latch.LatchNeg0 <-> Latch/LatchNeg0
//     PlcTask Inputs/GVL_iXlinker.EtherCAT_Master_ERxxxx.Beckhoff_ER1xxx.Beckhoff_ER1xxxEK1122.A_0008_ER1258_0001_0019.Latch.LatchNeg1 <-> Latch/LatchNeg1
//     PlcTask Inputs/GVL_iXlinker.EtherCAT_Master_ERxxxx.Beckhoff_ER1xxx.Beckhoff_ER1xxxEK1122.A_0008_ER1258_0001_0019.WcState.WcState0 <-> WcState/WcState0
//     PlcTask Inputs/GVL_iXlinker.EtherCAT_Master_ERxxxx.Beckhoff_ER1xxx.Beckhoff_ER1xxxEK1122.A_0008_ER1258_0001_0019.WcState.WcState1 <-> WcState/WcState1
//     PlcTask Inputs/GVL_iXlinker.EtherCAT_Master_ERxxxx.Beckhoff_ER1xxx.Beckhoff_ER1xxxEK1122.A_0008_ER1258_0001_0019.WcState.InputToggle0 <-> WcState/InputToggle0
//     PlcTask Inputs/GVL_iXlinker.EtherCAT_Master_ERxxxx.Beckhoff_ER1xxx.Beckhoff_ER1xxxEK1122.A_0008_ER1258_0001_0019.WcState.InputToggle1 <-> WcState/InputToggle1
//     PlcTask Inputs/GVL_iXlinker.EtherCAT_Master_ERxxxx.Beckhoff_ER1xxx.Beckhoff_ER1xxxEK1122.A_0008_ER1258_0001_0019.InfoData.DcOutputShift <-> InfoData/DcOutputShift
//     PlcTask Inputs/GVL_iXlinker.EtherCAT_Master_ERxxxx.Beckhoff_ER1xxx.Beckhoff_ER1xxxEK1122.A_0008_ER1258_0001_0019.InfoData.DcInputShift <-> InfoData/DcInputShift
//     PlcTask Inputs/GVL_iXlinker.EtherCAT_Master_ERxxxx.Beckhoff_ER1xxx.Beckhoff_ER1xxxEK1122.A_0008_ER1258_0001_0019.InfoData.State <-> InfoData/State
//   PLC/PLC Instance <-> EtherCAT Master ERxxxx/Beckhoff ER1xxx/Beckhoff ER1xxxEK1122/A_0009(ER1258-0001-0020)
//     PlcTask Inputs/GVL_iXlinker.EtherCAT_Master_ERxxxx.Beckhoff_ER1xxx.Beckhoff_ER1xxxEK1122.A_0009_ER1258_0001_0020.Channel_1.Input <-> Channel 1/Input
//     PlcTask Inputs/GVL_iXlinker.EtherCAT_Master_ERxxxx.Beckhoff_ER1xxx.Beckhoff_ER1xxxEK1122.A_0009_ER1258_0001_0020.Channel_2.Input <-> Channel 2/Input
//     PlcTask Inputs/GVL_iXlinker.EtherCAT_Master_ERxxxx.Beckhoff_ER1xxx.Beckhoff_ER1xxxEK1122.A_0009_ER1258_0001_0020.Channel_3.Input <-> Channel 3/Input
//     PlcTask Inputs/GVL_iXlinker.EtherCAT_Master_ERxxxx.Beckhoff_ER1xxx.Beckhoff_ER1xxxEK1122.A_0009_ER1258_0001_0020.Channel_4.Input <-> Channel 4/Input
//     PlcTask Inputs/GVL_iXlinker.EtherCAT_Master_ERxxxx.Beckhoff_ER1xxx.Beckhoff_ER1xxxEK1122.A_0009_ER1258_0001_0020.Channel_5.Input <-> Channel 5/Input
//     PlcTask Inputs/GVL_iXlinker.EtherCAT_Master_ERxxxx.Beckhoff_ER1xxx.Beckhoff_ER1xxxEK1122.A_0009_ER1258_0001_0020.Channel_6.Input <-> Channel 6/Input
//     PlcTask Inputs/GVL_iXlinker.EtherCAT_Master_ERxxxx.Beckhoff_ER1xxx.Beckhoff_ER1xxxEK1122.A_0009_ER1258_0001_0020.Channel_7.Input <-> Channel 7/Input
//     PlcTask Inputs/GVL_iXlinker.EtherCAT_Master_ERxxxx.Beckhoff_ER1xxx.Beckhoff_ER1xxxEK1122.A_0009_ER1258_0001_0020.Channel_8.Input <-> Channel 8/Input
//     PlcTask Inputs/GVL_iXlinker.EtherCAT_Master_ERxxxx.Beckhoff_ER1xxx.Beckhoff_ER1xxxEK1122.A_0009_ER1258_0001_0020.Latch.Status0 <-> Latch/Status0
//     PlcTask Inputs/GVL_iXlinker.EtherCAT_Master_ERxxxx.Beckhoff_ER1xxx.Beckhoff_ER1xxxEK1122.A_0009_ER1258_0001_0020.Latch.Status1 <-> Latch/Status1
//     PlcTask Inputs/GVL_iXlinker.EtherCAT_Master_ERxxxx.Beckhoff_ER1xxx.Beckhoff_ER1xxxEK1122.A_0009_ER1258_0001_0020.Latch.LatchPos0 <-> Latch/LatchPos0
//     PlcTask Inputs/GVL_iXlinker.EtherCAT_Master_ERxxxx.Beckhoff_ER1xxx.Beckhoff_ER1xxxEK1122.A_0009_ER1258_0001_0020.Latch.LatchPos1 <-> Latch/LatchPos1
//     PlcTask Inputs/GVL_iXlinker.EtherCAT_Master_ERxxxx.Beckhoff_ER1xxx.Beckhoff_ER1xxxEK1122.A_0009_ER1258_0001_0020.Latch.LatchNeg0 <-> Latch/LatchNeg0
//     PlcTask Inputs/GVL_iXlinker.EtherCAT_Master_ERxxxx.Beckhoff_ER1xxx.Beckhoff_ER1xxxEK1122.A_0009_ER1258_0001_0020.Latch.LatchNeg1 <-> Latch/LatchNeg1
//     PlcTask Inputs/GVL_iXlinker.EtherCAT_Master_ERxxxx.Beckhoff_ER1xxx.Beckhoff_ER1xxxEK1122.A_0009_ER1258_0001_0020.WcState.WcState0 <-> WcState/WcState0
//     PlcTask Inputs/GVL_iXlinker.EtherCAT_Master_ERxxxx.Beckhoff_ER1xxx.Beckhoff_ER1xxxEK1122.A_0009_ER1258_0001_0020.WcState.WcState1 <-> WcState/WcState1
//     PlcTask Inputs/GVL_iXlinker.EtherCAT_Master_ERxxxx.Beckhoff_ER1xxx.Beckhoff_ER1xxxEK1122.A_0009_ER1258_0001_0020.WcState.InputToggle0 <-> WcState/InputToggle0
//     PlcTask Inputs/GVL_iXlinker.EtherCAT_Master_ERxxxx.Beckhoff_ER1xxx.Beckhoff_ER1xxxEK1122.A_0009_ER1258_0001_0020.WcState.InputToggle1 <-> WcState/InputToggle1
//     PlcTask Inputs/GVL_iXlinker.EtherCAT_Master_ERxxxx.Beckhoff_ER1xxx.Beckhoff_ER1xxxEK1122.A_0009_ER1258_0001_0020.InfoData.DcOutputShift <-> InfoData/DcOutputShift
//     PlcTask Inputs/GVL_iXlinker.EtherCAT_Master_ERxxxx.Beckhoff_ER1xxx.Beckhoff_ER1xxxEK1122.A_0009_ER1258_0001_0020.InfoData.DcInputShift <-> InfoData/DcInputShift
//     PlcTask Inputs/GVL_iXlinker.EtherCAT_Master_ERxxxx.Beckhoff_ER1xxx.Beckhoff_ER1xxxEK1122.A_0009_ER1258_0001_0020.InfoData.State <-> InfoData/State
//   PLC/PLC Instance <-> EtherCAT Master ERxxxx/Beckhoff ER1xxx/Beckhoff ER1xxxEK1122/A_0010(ER1258-0002-0019)
//     PlcTask Inputs/GVL_iXlinker.EtherCAT_Master_ERxxxx.Beckhoff_ER1xxx.Beckhoff_ER1xxxEK1122.A_0010_ER1258_0002_0019.Channel_1.Input <-> Channel 1/Input
//     PlcTask Inputs/GVL_iXlinker.EtherCAT_Master_ERxxxx.Beckhoff_ER1xxx.Beckhoff_ER1xxxEK1122.A_0010_ER1258_0002_0019.Channel_2.Input <-> Channel 2/Input
//     PlcTask Inputs/GVL_iXlinker.EtherCAT_Master_ERxxxx.Beckhoff_ER1xxx.Beckhoff_ER1xxxEK1122.A_0010_ER1258_0002_0019.Channel_3.Input <-> Channel 3/Input
//     PlcTask Inputs/GVL_iXlinker.EtherCAT_Master_ERxxxx.Beckhoff_ER1xxx.Beckhoff_ER1xxxEK1122.A_0010_ER1258_0002_0019.Channel_4.Input <-> Channel 4/Input
//     PlcTask Inputs/GVL_iXlinker.EtherCAT_Master_ERxxxx.Beckhoff_ER1xxx.Beckhoff_ER1xxxEK1122.A_0010_ER1258_0002_0019.Channel_5.Input <-> Channel 5/Input
//     PlcTask Inputs/GVL_iXlinker.EtherCAT_Master_ERxxxx.Beckhoff_ER1xxx.Beckhoff_ER1xxxEK1122.A_0010_ER1258_0002_0019.Channel_6.Input <-> Channel 6/Input
//     PlcTask Inputs/GVL_iXlinker.EtherCAT_Master_ERxxxx.Beckhoff_ER1xxx.Beckhoff_ER1xxxEK1122.A_0010_ER1258_0002_0019.Channel_7.Input <-> Channel 7/Input
//     PlcTask Inputs/GVL_iXlinker.EtherCAT_Master_ERxxxx.Beckhoff_ER1xxx.Beckhoff_ER1xxxEK1122.A_0010_ER1258_0002_0019.Channel_8.Input <-> Channel 8/Input
//     PlcTask Inputs/GVL_iXlinker.EtherCAT_Master_ERxxxx.Beckhoff_ER1xxx.Beckhoff_ER1xxxEK1122.A_0010_ER1258_0002_0019.Latch.Status0 <-> Latch/Status0
//     PlcTask Inputs/GVL_iXlinker.EtherCAT_Master_ERxxxx.Beckhoff_ER1xxx.Beckhoff_ER1xxxEK1122.A_0010_ER1258_0002_0019.Latch.Status1 <-> Latch/Status1
//     PlcTask Inputs/GVL_iXlinker.EtherCAT_Master_ERxxxx.Beckhoff_ER1xxx.Beckhoff_ER1xxxEK1122.A_0010_ER1258_0002_0019.Latch.LatchPos0 <-> Latch/LatchPos0
//     PlcTask Inputs/GVL_iXlinker.EtherCAT_Master_ERxxxx.Beckhoff_ER1xxx.Beckhoff_ER1xxxEK1122.A_0010_ER1258_0002_0019.Latch.LatchPos1 <-> Latch/LatchPos1
//     PlcTask Inputs/GVL_iXlinker.EtherCAT_Master_ERxxxx.Beckhoff_ER1xxx.Beckhoff_ER1xxxEK1122.A_0010_ER1258_0002_0019.Latch.LatchNeg0 <-> Latch/LatchNeg0
//     PlcTask Inputs/GVL_iXlinker.EtherCAT_Master_ERxxxx.Beckhoff_ER1xxx.Beckhoff_ER1xxxEK1122.A_0010_ER1258_0002_0019.Latch.LatchNeg1 <-> Latch/LatchNeg1
//     PlcTask Inputs/GVL_iXlinker.EtherCAT_Master_ERxxxx.Beckhoff_ER1xxx.Beckhoff_ER1xxxEK1122.A_0010_ER1258_0002_0019.WcState.WcState0 <-> WcState/WcState0
//     PlcTask Inputs/GVL_iXlinker.EtherCAT_Master_ERxxxx.Beckhoff_ER1xxx.Beckhoff_ER1xxxEK1122.A_0010_ER1258_0002_0019.WcState.WcState1 <-> WcState/WcState1
//     PlcTask Inputs/GVL_iXlinker.EtherCAT_Master_ERxxxx.Beckhoff_ER1xxx.Beckhoff_ER1xxxEK1122.A_0010_ER1258_0002_0019.WcState.InputToggle0 <-> WcState/InputToggle0
//     PlcTask Inputs/GVL_iXlinker.EtherCAT_Master_ERxxxx.Beckhoff_ER1xxx.Beckhoff_ER1xxxEK1122.A_0010_ER1258_0002_0019.WcState.InputToggle1 <-> WcState/InputToggle1
//     PlcTask Inputs/GVL_iXlinker.EtherCAT_Master_ERxxxx.Beckhoff_ER1xxx.Beckhoff_ER1xxxEK1122.A_0010_ER1258_0002_0019.InfoData.DcOutputShift <-> InfoData/DcOutputShift
//     PlcTask Inputs/GVL_iXlinker.EtherCAT_Master_ERxxxx.Beckhoff_ER1xxx.Beckhoff_ER1xxxEK1122.A_0010_ER1258_0002_0019.InfoData.DcInputShift <-> InfoData/DcInputShift
//     PlcTask Inputs/GVL_iXlinker.EtherCAT_Master_ERxxxx.Beckhoff_ER1xxx.Beckhoff_ER1xxxEK1122.A_0010_ER1258_0002_0019.InfoData.State <-> InfoData/State
//   PLC/PLC Instance <-> EtherCAT Master ERxxxx/Beckhoff ER1xxx/Beckhoff ER1xxxEK1122/A_0011(ER1258-0002-0020)
//     PlcTask Inputs/GVL_iXlinker.EtherCAT_Master_ERxxxx.Beckhoff_ER1xxx.Beckhoff_ER1xxxEK1122.A_0011_ER1258_0002_0020.Channel_1.Input <-> Channel 1/Input
//     PlcTask Inputs/GVL_iXlinker.EtherCAT_Master_ERxxxx.Beckhoff_ER1xxx.Beckhoff_ER1xxxEK1122.A_0011_ER1258_0002_0020.Channel_2.Input <-> Channel 2/Input
//     PlcTask Inputs/GVL_iXlinker.EtherCAT_Master_ERxxxx.Beckhoff_ER1xxx.Beckhoff_ER1xxxEK1122.A_0011_ER1258_0002_0020.Channel_3.Input <-> Channel 3/Input
//     PlcTask Inputs/GVL_iXlinker.EtherCAT_Master_ERxxxx.Beckhoff_ER1xxx.Beckhoff_ER1xxxEK1122.A_0011_ER1258_0002_0020.Channel_4.Input <-> Channel 4/Input
//     PlcTask Inputs/GVL_iXlinker.EtherCAT_Master_ERxxxx.Beckhoff_ER1xxx.Beckhoff_ER1xxxEK1122.A_0011_ER1258_0002_0020.Channel_5.Input <-> Channel 5/Input
//     PlcTask Inputs/GVL_iXlinker.EtherCAT_Master_ERxxxx.Beckhoff_ER1xxx.Beckhoff_ER1xxxEK1122.A_0011_ER1258_0002_0020.Channel_6.Input <-> Channel 6/Input
//     PlcTask Inputs/GVL_iXlinker.EtherCAT_Master_ERxxxx.Beckhoff_ER1xxx.Beckhoff_ER1xxxEK1122.A_0011_ER1258_0002_0020.Channel_7.Input <-> Channel 7/Input
//     PlcTask Inputs/GVL_iXlinker.EtherCAT_Master_ERxxxx.Beckhoff_ER1xxx.Beckhoff_ER1xxxEK1122.A_0011_ER1258_0002_0020.Channel_8.Input <-> Channel 8/Input
//     PlcTask Inputs/GVL_iXlinker.EtherCAT_Master_ERxxxx.Beckhoff_ER1xxx.Beckhoff_ER1xxxEK1122.A_0011_ER1258_0002_0020.Latch.Status0 <-> Latch/Status0
//     PlcTask Inputs/GVL_iXlinker.EtherCAT_Master_ERxxxx.Beckhoff_ER1xxx.Beckhoff_ER1xxxEK1122.A_0011_ER1258_0002_0020.Latch.Status1 <-> Latch/Status1
//     PlcTask Inputs/GVL_iXlinker.EtherCAT_Master_ERxxxx.Beckhoff_ER1xxx.Beckhoff_ER1xxxEK1122.A_0011_ER1258_0002_0020.Latch.LatchPos0 <-> Latch/LatchPos0
//     PlcTask Inputs/GVL_iXlinker.EtherCAT_Master_ERxxxx.Beckhoff_ER1xxx.Beckhoff_ER1xxxEK1122.A_0011_ER1258_0002_0020.Latch.LatchPos1 <-> Latch/LatchPos1
//     PlcTask Inputs/GVL_iXlinker.EtherCAT_Master_ERxxxx.Beckhoff_ER1xxx.Beckhoff_ER1xxxEK1122.A_0011_ER1258_0002_0020.Latch.LatchNeg0 <-> Latch/LatchNeg0
//     PlcTask Inputs/GVL_iXlinker.EtherCAT_Master_ERxxxx.Beckhoff_ER1xxx.Beckhoff_ER1xxxEK1122.A_0011_ER1258_0002_0020.Latch.LatchNeg1 <-> Latch/LatchNeg1
//     PlcTask Inputs/GVL_iXlinker.EtherCAT_Master_ERxxxx.Beckhoff_ER1xxx.Beckhoff_ER1xxxEK1122.A_0011_ER1258_0002_0020.WcState.WcState0 <-> WcState/WcState0
//     PlcTask Inputs/GVL_iXlinker.EtherCAT_Master_ERxxxx.Beckhoff_ER1xxx.Beckhoff_ER1xxxEK1122.A_0011_ER1258_0002_0020.WcState.WcState1 <-> WcState/WcState1
//     PlcTask Inputs/GVL_iXlinker.EtherCAT_Master_ERxxxx.Beckhoff_ER1xxx.Beckhoff_ER1xxxEK1122.A_0011_ER1258_0002_0020.WcState.InputToggle0 <-> WcState/InputToggle0
//     PlcTask Inputs/GVL_iXlinker.EtherCAT_Master_ERxxxx.Beckhoff_ER1xxx.Beckhoff_ER1xxxEK1122.A_0011_ER1258_0002_0020.WcState.InputToggle1 <-> WcState/InputToggle1
//     PlcTask Inputs/GVL_iXlinker.EtherCAT_Master_ERxxxx.Beckhoff_ER1xxx.Beckhoff_ER1xxxEK1122.A_0011_ER1258_0002_0020.InfoData.DcOutputShift <-> InfoData/DcOutputShift
//     PlcTask Inputs/GVL_iXlinker.EtherCAT_Master_ERxxxx.Beckhoff_ER1xxx.Beckhoff_ER1xxxEK1122.A_0011_ER1258_0002_0020.InfoData.DcInputShift <-> InfoData/DcInputShift
//     PlcTask Inputs/GVL_iXlinker.EtherCAT_Master_ERxxxx.Beckhoff_ER1xxx.Beckhoff_ER1xxxEK1122.A_0011_ER1258_0002_0020.InfoData.State <-> InfoData/State
//   PLC/PLC Instance <-> EtherCAT Master ERxxxx/Beckhoff ER1xxx/Beckhoff ER1xxxEK1122/A_0012(ER1518-0002-0018)
//     PlcTask Inputs/GVL_iXlinker.EtherCAT_Master_ERxxxx.Beckhoff_ER1xxx.Beckhoff_ER1xxxEK1122.A_0012_ER1518_0002_0018.CNT_Input_Channel_1.Status/Set_counter_done <-> CNT Input Channel 1/Status/Set counter done
//     PlcTask Inputs/GVL_iXlinker.EtherCAT_Master_ERxxxx.Beckhoff_ER1xxx.Beckhoff_ER1xxxEK1122.A_0012_ER1518_0002_0018.CNT_Input_Channel_2.Status/Set_counter_done <-> CNT Input Channel 2/Status/Set counter done
//     PlcTask Inputs/GVL_iXlinker.EtherCAT_Master_ERxxxx.Beckhoff_ER1xxx.Beckhoff_ER1xxxEK1122.A_0012_ER1518_0002_0018.CNT_Input_Channel_1.Status/Counter_inhibited <-> CNT Input Channel 1/Status/Counter inhibited
//     PlcTask Inputs/GVL_iXlinker.EtherCAT_Master_ERxxxx.Beckhoff_ER1xxx.Beckhoff_ER1xxxEK1122.A_0012_ER1518_0002_0018.CNT_Input_Channel_2.Status/Counter_inhibited <-> CNT Input Channel 2/Status/Counter inhibited
//     PlcTask Inputs/GVL_iXlinker.EtherCAT_Master_ERxxxx.Beckhoff_ER1xxx.Beckhoff_ER1xxxEK1122.A_0012_ER1518_0002_0018.CNT_Input_Channel_1.Status/Status_of_input_UD <-> CNT Input Channel 1/Status/Status of input UD
//     PlcTask Inputs/GVL_iXlinker.EtherCAT_Master_ERxxxx.Beckhoff_ER1xxx.Beckhoff_ER1xxxEK1122.A_0012_ER1518_0002_0018.CNT_Input_Channel_2.Status/Status_of_input_UD <-> CNT Input Channel 2/Status/Status of input UD
//     PlcTask Inputs/GVL_iXlinker.EtherCAT_Master_ERxxxx.Beckhoff_ER1xxx.Beckhoff_ER1xxxEK1122.A_0012_ER1518_0002_0018.CNT_Input_Channel_1.Status/Status_of_input_clock <-> CNT Input Channel 1/Status/Status of input clock
//     PlcTask Inputs/GVL_iXlinker.EtherCAT_Master_ERxxxx.Beckhoff_ER1xxx.Beckhoff_ER1xxxEK1122.A_0012_ER1518_0002_0018.CNT_Input_Channel_2.Status/Status_of_input_clock <-> CNT Input Channel 2/Status/Status of input clock
//     PlcTask Inputs/GVL_iXlinker.EtherCAT_Master_ERxxxx.Beckhoff_ER1xxx.Beckhoff_ER1xxxEK1122.A_0012_ER1518_0002_0018.CNT_Input_Channel_1.Status/Sync_error <-> CNT Input Channel 1/Status/Sync error
//     PlcTask Inputs/GVL_iXlinker.EtherCAT_Master_ERxxxx.Beckhoff_ER1xxx.Beckhoff_ER1xxxEK1122.A_0012_ER1518_0002_0018.CNT_Input_Channel_2.Status/Sync_error <-> CNT Input Channel 2/Status/Sync error
//     PlcTask Inputs/GVL_iXlinker.EtherCAT_Master_ERxxxx.Beckhoff_ER1xxx.Beckhoff_ER1xxxEK1122.A_0012_ER1518_0002_0018.CNT_Input_Channel_1.Status/TxPDO_State <-> CNT Input Channel 1/Status/TxPDO State
//     PlcTask Inputs/GVL_iXlinker.EtherCAT_Master_ERxxxx.Beckhoff_ER1xxx.Beckhoff_ER1xxxEK1122.A_0012_ER1518_0002_0018.CNT_Input_Channel_2.Status/TxPDO_State <-> CNT Input Channel 2/Status/TxPDO State
//     PlcTask Inputs/GVL_iXlinker.EtherCAT_Master_ERxxxx.Beckhoff_ER1xxx.Beckhoff_ER1xxxEK1122.A_0012_ER1518_0002_0018.CNT_Input_Channel_1.Status/TxPDO_Toggle <-> CNT Input Channel 1/Status/TxPDO Toggle
//     PlcTask Inputs/GVL_iXlinker.EtherCAT_Master_ERxxxx.Beckhoff_ER1xxx.Beckhoff_ER1xxxEK1122.A_0012_ER1518_0002_0018.CNT_Input_Channel_2.Status/TxPDO_Toggle <-> CNT Input Channel 2/Status/TxPDO Toggle
//     PlcTask Inputs/GVL_iXlinker.EtherCAT_Master_ERxxxx.Beckhoff_ER1xxx.Beckhoff_ER1xxxEK1122.A_0012_ER1518_0002_0018.CNT_Input_Channel_1.Counter_value <-> CNT Input Channel 1/Counter value
//     PlcTask Inputs/GVL_iXlinker.EtherCAT_Master_ERxxxx.Beckhoff_ER1xxx.Beckhoff_ER1xxxEK1122.A_0012_ER1518_0002_0018.CNT_Input_Channel_2.Counter_value <-> CNT Input Channel 2/Counter value
//     PlcTask Inputs/GVL_iXlinker.EtherCAT_Master_ERxxxx.Beckhoff_ER1xxx.Beckhoff_ER1xxxEK1122.A_0012_ER1518_0002_0018.DIG_Inputs.Input[0] <-> DIG Inputs/Input 0
//     PlcTask Inputs/GVL_iXlinker.EtherCAT_Master_ERxxxx.Beckhoff_ER1xxx.Beckhoff_ER1xxxEK1122.A_0012_ER1518_0002_0018.DIG_Inputs.Input[1] <-> DIG Inputs/Input 1
//     PlcTask Inputs/GVL_iXlinker.EtherCAT_Master_ERxxxx.Beckhoff_ER1xxx.Beckhoff_ER1xxxEK1122.A_0012_ER1518_0002_0018.DIG_Inputs.Input[2] <-> DIG Inputs/Input 2
//     PlcTask Inputs/GVL_iXlinker.EtherCAT_Master_ERxxxx.Beckhoff_ER1xxx.Beckhoff_ER1xxxEK1122.A_0012_ER1518_0002_0018.DIG_Inputs.Input[3] <-> DIG Inputs/Input 3
//     PlcTask Inputs/GVL_iXlinker.EtherCAT_Master_ERxxxx.Beckhoff_ER1xxx.Beckhoff_ER1xxxEK1122.A_0012_ER1518_0002_0018.DIG_Inputs.Input[4] <-> DIG Inputs/Input 4
//     PlcTask Inputs/GVL_iXlinker.EtherCAT_Master_ERxxxx.Beckhoff_ER1xxx.Beckhoff_ER1xxxEK1122.A_0012_ER1518_0002_0018.DIG_Inputs.Input[5] <-> DIG Inputs/Input 5
//     PlcTask Inputs/GVL_iXlinker.EtherCAT_Master_ERxxxx.Beckhoff_ER1xxx.Beckhoff_ER1xxxEK1122.A_0012_ER1518_0002_0018.DIG_Inputs.Input[6] <-> DIG Inputs/Input 6
//     PlcTask Inputs/GVL_iXlinker.EtherCAT_Master_ERxxxx.Beckhoff_ER1xxx.Beckhoff_ER1xxxEK1122.A_0012_ER1518_0002_0018.DIG_Inputs.Input[7] <-> DIG Inputs/Input 7
//     PlcTask Inputs/GVL_iXlinker.EtherCAT_Master_ERxxxx.Beckhoff_ER1xxx.Beckhoff_ER1xxxEK1122.A_0012_ER1518_0002_0018.DIG_Inputs_Device.Status/Error_channel_1 <-> DIG Inputs Device/Status/Error channel 1
//     PlcTask Inputs/GVL_iXlinker.EtherCAT_Master_ERxxxx.Beckhoff_ER1xxx.Beckhoff_ER1xxxEK1122.A_0012_ER1518_0002_0018.DIG_Inputs_Device.Status/Error_channel_2 <-> DIG Inputs Device/Status/Error channel 2
//     PlcTask Inputs/GVL_iXlinker.EtherCAT_Master_ERxxxx.Beckhoff_ER1xxx.Beckhoff_ER1xxxEK1122.A_0012_ER1518_0002_0018.DIG_Inputs_Device.Status/Sync_error <-> DIG Inputs Device/Status/Sync error
//     PlcTask Inputs/GVL_iXlinker.EtherCAT_Master_ERxxxx.Beckhoff_ER1xxx.Beckhoff_ER1xxxEK1122.A_0012_ER1518_0002_0018.DIG_Inputs_Device.Status/TxPDO_State <-> DIG Inputs Device/Status/TxPDO State
//     PlcTask Inputs/GVL_iXlinker.EtherCAT_Master_ERxxxx.Beckhoff_ER1xxx.Beckhoff_ER1xxxEK1122.A_0012_ER1518_0002_0018.DIG_Inputs_Device.Status/TxPDO_Toggle <-> DIG Inputs Device/Status/TxPDO Toggle
//     PlcTask Outputs/GVL_iXlinker.EtherCAT_Master_ERxxxx.Beckhoff_ER1xxx.Beckhoff_ER1xxxEK1122.A_0012_ER1518_0002_0018.CNT_Output_Channel_1.Control/Set_counter <-> CNT Output Channel 1/Control/Set counter
//     PlcTask Outputs/GVL_iXlinker.EtherCAT_Master_ERxxxx.Beckhoff_ER1xxx.Beckhoff_ER1xxxEK1122.A_0012_ER1518_0002_0018.CNT_Output_Channel_2.Control/Set_counter <-> CNT Output Channel 2/Control/Set counter
//     PlcTask Outputs/GVL_iXlinker.EtherCAT_Master_ERxxxx.Beckhoff_ER1xxx.Beckhoff_ER1xxxEK1122.A_0012_ER1518_0002_0018.CNT_Output_Channel_1.Control/Inhibit_counter <-> CNT Output Channel 1/Control/Inhibit counter
//     PlcTask Outputs/GVL_iXlinker.EtherCAT_Master_ERxxxx.Beckhoff_ER1xxx.Beckhoff_ER1xxxEK1122.A_0012_ER1518_0002_0018.CNT_Output_Channel_2.Control/Inhibit_counter <-> CNT Output Channel 2/Control/Inhibit counter
//     PlcTask Outputs/GVL_iXlinker.EtherCAT_Master_ERxxxx.Beckhoff_ER1xxx.Beckhoff_ER1xxxEK1122.A_0012_ER1518_0002_0018.CNT_Output_Channel_1.Set_counter_value <-> CNT Output Channel 1/Set counter value
//     PlcTask Outputs/GVL_iXlinker.EtherCAT_Master_ERxxxx.Beckhoff_ER1xxx.Beckhoff_ER1xxxEK1122.A_0012_ER1518_0002_0018.CNT_Output_Channel_2.Set_counter_value <-> CNT Output Channel 2/Set counter value
//     PlcTask Inputs/GVL_iXlinker.EtherCAT_Master_ERxxxx.Beckhoff_ER1xxx.Beckhoff_ER1xxxEK1122.A_0012_ER1518_0002_0018.WcState.WcState <-> WcState/WcState
//     PlcTask Inputs/GVL_iXlinker.EtherCAT_Master_ERxxxx.Beckhoff_ER1xxx.Beckhoff_ER1xxxEK1122.A_0012_ER1518_0002_0018.WcState.InputToggle <-> WcState/InputToggle
//     PlcTask Inputs/GVL_iXlinker.EtherCAT_Master_ERxxxx.Beckhoff_ER1xxx.Beckhoff_ER1xxxEK1122.A_0012_ER1518_0002_0018.InfoData.AdsAddr <-> InfoData/AdsAddr
//     PlcTask Inputs/GVL_iXlinker.EtherCAT_Master_ERxxxx.Beckhoff_ER1xxx.Beckhoff_ER1xxxEK1122.A_0012_ER1518_0002_0018.InfoData.State <-> InfoData/State
//   PLC/PLC Instance <-> EtherCAT Master ERxxxx/Beckhoff ER1xxx/Beckhoff ER1xxxEK1122/A_0013(ER1518-0002-0019)
//     PlcTask Inputs/GVL_iXlinker.EtherCAT_Master_ERxxxx.Beckhoff_ER1xxx.Beckhoff_ER1xxxEK1122.A_0013_ER1518_0002_0019.CNT_Input_Channel_1.Status/Set_counter_done <-> CNT Input Channel 1/Status/Set counter done
//     PlcTask Inputs/GVL_iXlinker.EtherCAT_Master_ERxxxx.Beckhoff_ER1xxx.Beckhoff_ER1xxxEK1122.A_0013_ER1518_0002_0019.CNT_Input_Channel_2.Status/Set_counter_done <-> CNT Input Channel 2/Status/Set counter done
//     PlcTask Inputs/GVL_iXlinker.EtherCAT_Master_ERxxxx.Beckhoff_ER1xxx.Beckhoff_ER1xxxEK1122.A_0013_ER1518_0002_0019.CNT_Input_Channel_1.Status/Counter_inhibited <-> CNT Input Channel 1/Status/Counter inhibited
//     PlcTask Inputs/GVL_iXlinker.EtherCAT_Master_ERxxxx.Beckhoff_ER1xxx.Beckhoff_ER1xxxEK1122.A_0013_ER1518_0002_0019.CNT_Input_Channel_2.Status/Counter_inhibited <-> CNT Input Channel 2/Status/Counter inhibited
//     PlcTask Inputs/GVL_iXlinker.EtherCAT_Master_ERxxxx.Beckhoff_ER1xxx.Beckhoff_ER1xxxEK1122.A_0013_ER1518_0002_0019.CNT_Input_Channel_1.Status/Status_of_input_UD <-> CNT Input Channel 1/Status/Status of input UD
//     PlcTask Inputs/GVL_iXlinker.EtherCAT_Master_ERxxxx.Beckhoff_ER1xxx.Beckhoff_ER1xxxEK1122.A_0013_ER1518_0002_0019.CNT_Input_Channel_2.Status/Status_of_input_UD <-> CNT Input Channel 2/Status/Status of input UD
//     PlcTask Inputs/GVL_iXlinker.EtherCAT_Master_ERxxxx.Beckhoff_ER1xxx.Beckhoff_ER1xxxEK1122.A_0013_ER1518_0002_0019.CNT_Input_Channel_1.Status/Status_of_input_clock <-> CNT Input Channel 1/Status/Status of input clock
//     PlcTask Inputs/GVL_iXlinker.EtherCAT_Master_ERxxxx.Beckhoff_ER1xxx.Beckhoff_ER1xxxEK1122.A_0013_ER1518_0002_0019.CNT_Input_Channel_2.Status/Status_of_input_clock <-> CNT Input Channel 2/Status/Status of input clock
//     PlcTask Inputs/GVL_iXlinker.EtherCAT_Master_ERxxxx.Beckhoff_ER1xxx.Beckhoff_ER1xxxEK1122.A_0013_ER1518_0002_0019.CNT_Input_Channel_1.Status/Sync_error <-> CNT Input Channel 1/Status/Sync error
//     PlcTask Inputs/GVL_iXlinker.EtherCAT_Master_ERxxxx.Beckhoff_ER1xxx.Beckhoff_ER1xxxEK1122.A_0013_ER1518_0002_0019.CNT_Input_Channel_2.Status/Sync_error <-> CNT Input Channel 2/Status/Sync error
//     PlcTask Inputs/GVL_iXlinker.EtherCAT_Master_ERxxxx.Beckhoff_ER1xxx.Beckhoff_ER1xxxEK1122.A_0013_ER1518_0002_0019.CNT_Input_Channel_1.Status/TxPDO_State <-> CNT Input Channel 1/Status/TxPDO State
//     PlcTask Inputs/GVL_iXlinker.EtherCAT_Master_ERxxxx.Beckhoff_ER1xxx.Beckhoff_ER1xxxEK1122.A_0013_ER1518_0002_0019.CNT_Input_Channel_2.Status/TxPDO_State <-> CNT Input Channel 2/Status/TxPDO State
//     PlcTask Inputs/GVL_iXlinker.EtherCAT_Master_ERxxxx.Beckhoff_ER1xxx.Beckhoff_ER1xxxEK1122.A_0013_ER1518_0002_0019.CNT_Input_Channel_1.Status/TxPDO_Toggle <-> CNT Input Channel 1/Status/TxPDO Toggle
//     PlcTask Inputs/GVL_iXlinker.EtherCAT_Master_ERxxxx.Beckhoff_ER1xxx.Beckhoff_ER1xxxEK1122.A_0013_ER1518_0002_0019.CNT_Input_Channel_2.Status/TxPDO_Toggle <-> CNT Input Channel 2/Status/TxPDO Toggle
//     PlcTask Inputs/GVL_iXlinker.EtherCAT_Master_ERxxxx.Beckhoff_ER1xxx.Beckhoff_ER1xxxEK1122.A_0013_ER1518_0002_0019.CNT_Input_Channel_1.Counter_value <-> CNT Input Channel 1/Counter value
//     PlcTask Inputs/GVL_iXlinker.EtherCAT_Master_ERxxxx.Beckhoff_ER1xxx.Beckhoff_ER1xxxEK1122.A_0013_ER1518_0002_0019.CNT_Input_Channel_2.Counter_value <-> CNT Input Channel 2/Counter value
//     PlcTask Inputs/GVL_iXlinker.EtherCAT_Master_ERxxxx.Beckhoff_ER1xxx.Beckhoff_ER1xxxEK1122.A_0013_ER1518_0002_0019.DIG_Inputs.Input[0] <-> DIG Inputs/Input 0
//     PlcTask Inputs/GVL_iXlinker.EtherCAT_Master_ERxxxx.Beckhoff_ER1xxx.Beckhoff_ER1xxxEK1122.A_0013_ER1518_0002_0019.DIG_Inputs.Input[1] <-> DIG Inputs/Input 1
//     PlcTask Inputs/GVL_iXlinker.EtherCAT_Master_ERxxxx.Beckhoff_ER1xxx.Beckhoff_ER1xxxEK1122.A_0013_ER1518_0002_0019.DIG_Inputs.Input[2] <-> DIG Inputs/Input 2
//     PlcTask Inputs/GVL_iXlinker.EtherCAT_Master_ERxxxx.Beckhoff_ER1xxx.Beckhoff_ER1xxxEK1122.A_0013_ER1518_0002_0019.DIG_Inputs.Input[3] <-> DIG Inputs/Input 3
//     PlcTask Inputs/GVL_iXlinker.EtherCAT_Master_ERxxxx.Beckhoff_ER1xxx.Beckhoff_ER1xxxEK1122.A_0013_ER1518_0002_0019.DIG_Inputs.Input[4] <-> DIG Inputs/Input 4
//     PlcTask Inputs/GVL_iXlinker.EtherCAT_Master_ERxxxx.Beckhoff_ER1xxx.Beckhoff_ER1xxxEK1122.A_0013_ER1518_0002_0019.DIG_Inputs.Input[5] <-> DIG Inputs/Input 5
//     PlcTask Inputs/GVL_iXlinker.EtherCAT_Master_ERxxxx.Beckhoff_ER1xxx.Beckhoff_ER1xxxEK1122.A_0013_ER1518_0002_0019.DIG_Inputs.Input[6] <-> DIG Inputs/Input 6
//     PlcTask Inputs/GVL_iXlinker.EtherCAT_Master_ERxxxx.Beckhoff_ER1xxx.Beckhoff_ER1xxxEK1122.A_0013_ER1518_0002_0019.DIG_Inputs.Input[7] <-> DIG Inputs/Input 7
//     PlcTask Inputs/GVL_iXlinker.EtherCAT_Master_ERxxxx.Beckhoff_ER1xxx.Beckhoff_ER1xxxEK1122.A_0013_ER1518_0002_0019.DIG_Inputs_Device.Status/Error_channel_1 <-> DIG Inputs Device/Status/Error channel 1
//     PlcTask Inputs/GVL_iXlinker.EtherCAT_Master_ERxxxx.Beckhoff_ER1xxx.Beckhoff_ER1xxxEK1122.A_0013_ER1518_0002_0019.DIG_Inputs_Device.Status/Error_channel_2 <-> DIG Inputs Device/Status/Error channel 2
//     PlcTask Inputs/GVL_iXlinker.EtherCAT_Master_ERxxxx.Beckhoff_ER1xxx.Beckhoff_ER1xxxEK1122.A_0013_ER1518_0002_0019.DIG_Inputs_Device.Status/Sync_error <-> DIG Inputs Device/Status/Sync error
//     PlcTask Inputs/GVL_iXlinker.EtherCAT_Master_ERxxxx.Beckhoff_ER1xxx.Beckhoff_ER1xxxEK1122.A_0013_ER1518_0002_0019.DIG_Inputs_Device.Status/TxPDO_State <-> DIG Inputs Device/Status/TxPDO State
//     PlcTask Inputs/GVL_iXlinker.EtherCAT_Master_ERxxxx.Beckhoff_ER1xxx.Beckhoff_ER1xxxEK1122.A_0013_ER1518_0002_0019.DIG_Inputs_Device.Status/TxPDO_Toggle <-> DIG Inputs Device/Status/TxPDO Toggle
//     PlcTask Outputs/GVL_iXlinker.EtherCAT_Master_ERxxxx.Beckhoff_ER1xxx.Beckhoff_ER1xxxEK1122.A_0013_ER1518_0002_0019.CNT_Output_Channel_1.Control/Set_counter <-> CNT Output Channel 1/Control/Set counter
//     PlcTask Outputs/GVL_iXlinker.EtherCAT_Master_ERxxxx.Beckhoff_ER1xxx.Beckhoff_ER1xxxEK1122.A_0013_ER1518_0002_0019.CNT_Output_Channel_2.Control/Set_counter <-> CNT Output Channel 2/Control/Set counter
//     PlcTask Outputs/GVL_iXlinker.EtherCAT_Master_ERxxxx.Beckhoff_ER1xxx.Beckhoff_ER1xxxEK1122.A_0013_ER1518_0002_0019.CNT_Output_Channel_1.Control/Inhibit_counter <-> CNT Output Channel 1/Control/Inhibit counter
//     PlcTask Outputs/GVL_iXlinker.EtherCAT_Master_ERxxxx.Beckhoff_ER1xxx.Beckhoff_ER1xxxEK1122.A_0013_ER1518_0002_0019.CNT_Output_Channel_2.Control/Inhibit_counter <-> CNT Output Channel 2/Control/Inhibit counter
//     PlcTask Outputs/GVL_iXlinker.EtherCAT_Master_ERxxxx.Beckhoff_ER1xxx.Beckhoff_ER1xxxEK1122.A_0013_ER1518_0002_0019.CNT_Output_Channel_1.Set_counter_value <-> CNT Output Channel 1/Set counter value
//     PlcTask Outputs/GVL_iXlinker.EtherCAT_Master_ERxxxx.Beckhoff_ER1xxx.Beckhoff_ER1xxxEK1122.A_0013_ER1518_0002_0019.CNT_Output_Channel_2.Set_counter_value <-> CNT Output Channel 2/Set counter value
//     PlcTask Inputs/GVL_iXlinker.EtherCAT_Master_ERxxxx.Beckhoff_ER1xxx.Beckhoff_ER1xxxEK1122.A_0013_ER1518_0002_0019.WcState.WcState <-> WcState/WcState
//     PlcTask Inputs/GVL_iXlinker.EtherCAT_Master_ERxxxx.Beckhoff_ER1xxx.Beckhoff_ER1xxxEK1122.A_0013_ER1518_0002_0019.WcState.InputToggle <-> WcState/InputToggle
//     PlcTask Inputs/GVL_iXlinker.EtherCAT_Master_ERxxxx.Beckhoff_ER1xxx.Beckhoff_ER1xxxEK1122.A_0013_ER1518_0002_0019.InfoData.AdsAddr <-> InfoData/AdsAddr
//     PlcTask Inputs/GVL_iXlinker.EtherCAT_Master_ERxxxx.Beckhoff_ER1xxx.Beckhoff_ER1xxxEK1122.A_0013_ER1518_0002_0019.InfoData.State <-> InfoData/State
//   PLC/PLC Instance <-> EtherCAT Master ERxxxx/Beckhoff ER1xxx/Beckhoff ER1xxxEK1122/A_0014(ER1809-0021-0017)
//     PlcTask Inputs/GVL_iXlinker.EtherCAT_Master_ERxxxx.Beckhoff_ER1xxx.Beckhoff_ER1xxxEK1122.A_0014_ER1809_0021_0017.Channel_1.Input <-> Channel 1/Input
//     PlcTask Inputs/GVL_iXlinker.EtherCAT_Master_ERxxxx.Beckhoff_ER1xxx.Beckhoff_ER1xxxEK1122.A_0014_ER1809_0021_0017.Channel_2.Input <-> Channel 2/Input
//     PlcTask Inputs/GVL_iXlinker.EtherCAT_Master_ERxxxx.Beckhoff_ER1xxx.Beckhoff_ER1xxxEK1122.A_0014_ER1809_0021_0017.Channel_3.Input <-> Channel 3/Input
//     PlcTask Inputs/GVL_iXlinker.EtherCAT_Master_ERxxxx.Beckhoff_ER1xxx.Beckhoff_ER1xxxEK1122.A_0014_ER1809_0021_0017.Channel_4.Input <-> Channel 4/Input
//     PlcTask Inputs/GVL_iXlinker.EtherCAT_Master_ERxxxx.Beckhoff_ER1xxx.Beckhoff_ER1xxxEK1122.A_0014_ER1809_0021_0017.Channel_5.Input <-> Channel 5/Input
//     PlcTask Inputs/GVL_iXlinker.EtherCAT_Master_ERxxxx.Beckhoff_ER1xxx.Beckhoff_ER1xxxEK1122.A_0014_ER1809_0021_0017.Channel_6.Input <-> Channel 6/Input
//     PlcTask Inputs/GVL_iXlinker.EtherCAT_Master_ERxxxx.Beckhoff_ER1xxx.Beckhoff_ER1xxxEK1122.A_0014_ER1809_0021_0017.Channel_7.Input <-> Channel 7/Input
//     PlcTask Inputs/GVL_iXlinker.EtherCAT_Master_ERxxxx.Beckhoff_ER1xxx.Beckhoff_ER1xxxEK1122.A_0014_ER1809_0021_0017.Channel_8.Input <-> Channel 8/Input
//     PlcTask Inputs/GVL_iXlinker.EtherCAT_Master_ERxxxx.Beckhoff_ER1xxx.Beckhoff_ER1xxxEK1122.A_0014_ER1809_0021_0017.Channel_9.Input <-> Channel 9/Input
//     PlcTask Inputs/GVL_iXlinker.EtherCAT_Master_ERxxxx.Beckhoff_ER1xxx.Beckhoff_ER1xxxEK1122.A_0014_ER1809_0021_0017.Channel_10.Input <-> Channel 10/Input
//     PlcTask Inputs/GVL_iXlinker.EtherCAT_Master_ERxxxx.Beckhoff_ER1xxx.Beckhoff_ER1xxxEK1122.A_0014_ER1809_0021_0017.Channel_11.Input <-> Channel 11/Input
//     PlcTask Inputs/GVL_iXlinker.EtherCAT_Master_ERxxxx.Beckhoff_ER1xxx.Beckhoff_ER1xxxEK1122.A_0014_ER1809_0021_0017.Channel_12.Input <-> Channel 12/Input
//     PlcTask Inputs/GVL_iXlinker.EtherCAT_Master_ERxxxx.Beckhoff_ER1xxx.Beckhoff_ER1xxxEK1122.A_0014_ER1809_0021_0017.Channel_13.Input <-> Channel 13/Input
//     PlcTask Inputs/GVL_iXlinker.EtherCAT_Master_ERxxxx.Beckhoff_ER1xxx.Beckhoff_ER1xxxEK1122.A_0014_ER1809_0021_0017.Channel_14.Input <-> Channel 14/Input
//     PlcTask Inputs/GVL_iXlinker.EtherCAT_Master_ERxxxx.Beckhoff_ER1xxx.Beckhoff_ER1xxxEK1122.A_0014_ER1809_0021_0017.Channel_15.Input <-> Channel 15/Input
//     PlcTask Inputs/GVL_iXlinker.EtherCAT_Master_ERxxxx.Beckhoff_ER1xxx.Beckhoff_ER1xxxEK1122.A_0014_ER1809_0021_0017.Channel_16.Input <-> Channel 16/Input
//     PlcTask Inputs/GVL_iXlinker.EtherCAT_Master_ERxxxx.Beckhoff_ER1xxx.Beckhoff_ER1xxxEK1122.A_0014_ER1809_0021_0017.WcState.WcState <-> WcState/WcState
//     PlcTask Inputs/GVL_iXlinker.EtherCAT_Master_ERxxxx.Beckhoff_ER1xxx.Beckhoff_ER1xxxEK1122.A_0014_ER1809_0021_0017.WcState.InputToggle <-> WcState/InputToggle
//     PlcTask Inputs/GVL_iXlinker.EtherCAT_Master_ERxxxx.Beckhoff_ER1xxx.Beckhoff_ER1xxxEK1122.A_0014_ER1809_0021_0017.InfoData.State <-> InfoData/State
//   PLC/PLC Instance <-> EtherCAT Master ERxxxx/Beckhoff ER1xxx/Beckhoff ER1xxxEK1122/A_0015(ER1809-0022-0018)
//     PlcTask Inputs/GVL_iXlinker.EtherCAT_Master_ERxxxx.Beckhoff_ER1xxx.Beckhoff_ER1xxxEK1122.A_0015_ER1809_0022_0018.Channel_1.Input <-> Channel 1/Input
//     PlcTask Inputs/GVL_iXlinker.EtherCAT_Master_ERxxxx.Beckhoff_ER1xxx.Beckhoff_ER1xxxEK1122.A_0015_ER1809_0022_0018.Channel_2.Input <-> Channel 2/Input
//     PlcTask Inputs/GVL_iXlinker.EtherCAT_Master_ERxxxx.Beckhoff_ER1xxx.Beckhoff_ER1xxxEK1122.A_0015_ER1809_0022_0018.Channel_3.Input <-> Channel 3/Input
//     PlcTask Inputs/GVL_iXlinker.EtherCAT_Master_ERxxxx.Beckhoff_ER1xxx.Beckhoff_ER1xxxEK1122.A_0015_ER1809_0022_0018.Channel_4.Input <-> Channel 4/Input
//     PlcTask Inputs/GVL_iXlinker.EtherCAT_Master_ERxxxx.Beckhoff_ER1xxx.Beckhoff_ER1xxxEK1122.A_0015_ER1809_0022_0018.Channel_5.Input <-> Channel 5/Input
//     PlcTask Inputs/GVL_iXlinker.EtherCAT_Master_ERxxxx.Beckhoff_ER1xxx.Beckhoff_ER1xxxEK1122.A_0015_ER1809_0022_0018.Channel_6.Input <-> Channel 6/Input
//     PlcTask Inputs/GVL_iXlinker.EtherCAT_Master_ERxxxx.Beckhoff_ER1xxx.Beckhoff_ER1xxxEK1122.A_0015_ER1809_0022_0018.Channel_7.Input <-> Channel 7/Input
//     PlcTask Inputs/GVL_iXlinker.EtherCAT_Master_ERxxxx.Beckhoff_ER1xxx.Beckhoff_ER1xxxEK1122.A_0015_ER1809_0022_0018.Channel_8.Input <-> Channel 8/Input
//     PlcTask Inputs/GVL_iXlinker.EtherCAT_Master_ERxxxx.Beckhoff_ER1xxx.Beckhoff_ER1xxxEK1122.A_0015_ER1809_0022_0018.Channel_9.Input <-> Channel 9/Input
//     PlcTask Inputs/GVL_iXlinker.EtherCAT_Master_ERxxxx.Beckhoff_ER1xxx.Beckhoff_ER1xxxEK1122.A_0015_ER1809_0022_0018.Channel_10.Input <-> Channel 10/Input
//     PlcTask Inputs/GVL_iXlinker.EtherCAT_Master_ERxxxx.Beckhoff_ER1xxx.Beckhoff_ER1xxxEK1122.A_0015_ER1809_0022_0018.Channel_11.Input <-> Channel 11/Input
//     PlcTask Inputs/GVL_iXlinker.EtherCAT_Master_ERxxxx.Beckhoff_ER1xxx.Beckhoff_ER1xxxEK1122.A_0015_ER1809_0022_0018.Channel_12.Input <-> Channel 12/Input
//     PlcTask Inputs/GVL_iXlinker.EtherCAT_Master_ERxxxx.Beckhoff_ER1xxx.Beckhoff_ER1xxxEK1122.A_0015_ER1809_0022_0018.Channel_13.Input <-> Channel 13/Input
//     PlcTask Inputs/GVL_iXlinker.EtherCAT_Master_ERxxxx.Beckhoff_ER1xxx.Beckhoff_ER1xxxEK1122.A_0015_ER1809_0022_0018.Channel_14.Input <-> Channel 14/Input
//     PlcTask Inputs/GVL_iXlinker.EtherCAT_Master_ERxxxx.Beckhoff_ER1xxx.Beckhoff_ER1xxxEK1122.A_0015_ER1809_0022_0018.Channel_15.Input <-> Channel 15/Input
//     PlcTask Inputs/GVL_iXlinker.EtherCAT_Master_ERxxxx.Beckhoff_ER1xxx.Beckhoff_ER1xxxEK1122.A_0015_ER1809_0022_0018.Channel_16.Input <-> Channel 16/Input
//     PlcTask Inputs/GVL_iXlinker.EtherCAT_Master_ERxxxx.Beckhoff_ER1xxx.Beckhoff_ER1xxxEK1122.A_0015_ER1809_0022_0018.WcState.WcState <-> WcState/WcState
//     PlcTask Inputs/GVL_iXlinker.EtherCAT_Master_ERxxxx.Beckhoff_ER1xxx.Beckhoff_ER1xxxEK1122.A_0015_ER1809_0022_0018.WcState.InputToggle <-> WcState/InputToggle
//     PlcTask Inputs/GVL_iXlinker.EtherCAT_Master_ERxxxx.Beckhoff_ER1xxx.Beckhoff_ER1xxxEK1122.A_0015_ER1809_0022_0018.InfoData.State <-> InfoData/State
//   PLC/PLC Instance <-> EtherCAT Master ERxxxx/Beckhoff ER1xxx/Beckhoff ER1xxxEK1122/A_0016(ER1819-0021-0017)
//     PlcTask Inputs/GVL_iXlinker.EtherCAT_Master_ERxxxx.Beckhoff_ER1xxx.Beckhoff_ER1xxxEK1122.A_0016_ER1819_0021_0017.Channel_1.Input <-> Channel 1/Input
//     PlcTask Inputs/GVL_iXlinker.EtherCAT_Master_ERxxxx.Beckhoff_ER1xxx.Beckhoff_ER1xxxEK1122.A_0016_ER1819_0021_0017.Channel_2.Input <-> Channel 2/Input
//     PlcTask Inputs/GVL_iXlinker.EtherCAT_Master_ERxxxx.Beckhoff_ER1xxx.Beckhoff_ER1xxxEK1122.A_0016_ER1819_0021_0017.Channel_3.Input <-> Channel 3/Input
//     PlcTask Inputs/GVL_iXlinker.EtherCAT_Master_ERxxxx.Beckhoff_ER1xxx.Beckhoff_ER1xxxEK1122.A_0016_ER1819_0021_0017.Channel_4.Input <-> Channel 4/Input
//     PlcTask Inputs/GVL_iXlinker.EtherCAT_Master_ERxxxx.Beckhoff_ER1xxx.Beckhoff_ER1xxxEK1122.A_0016_ER1819_0021_0017.Channel_5.Input <-> Channel 5/Input
//     PlcTask Inputs/GVL_iXlinker.EtherCAT_Master_ERxxxx.Beckhoff_ER1xxx.Beckhoff_ER1xxxEK1122.A_0016_ER1819_0021_0017.Channel_6.Input <-> Channel 6/Input
//     PlcTask Inputs/GVL_iXlinker.EtherCAT_Master_ERxxxx.Beckhoff_ER1xxx.Beckhoff_ER1xxxEK1122.A_0016_ER1819_0021_0017.Channel_7.Input <-> Channel 7/Input
//     PlcTask Inputs/GVL_iXlinker.EtherCAT_Master_ERxxxx.Beckhoff_ER1xxx.Beckhoff_ER1xxxEK1122.A_0016_ER1819_0021_0017.Channel_8.Input <-> Channel 8/Input
//     PlcTask Inputs/GVL_iXlinker.EtherCAT_Master_ERxxxx.Beckhoff_ER1xxx.Beckhoff_ER1xxxEK1122.A_0016_ER1819_0021_0017.Channel_9.Input <-> Channel 9/Input
//     PlcTask Inputs/GVL_iXlinker.EtherCAT_Master_ERxxxx.Beckhoff_ER1xxx.Beckhoff_ER1xxxEK1122.A_0016_ER1819_0021_0017.Channel_10.Input <-> Channel 10/Input
//     PlcTask Inputs/GVL_iXlinker.EtherCAT_Master_ERxxxx.Beckhoff_ER1xxx.Beckhoff_ER1xxxEK1122.A_0016_ER1819_0021_0017.Channel_11.Input <-> Channel 11/Input
//     PlcTask Inputs/GVL_iXlinker.EtherCAT_Master_ERxxxx.Beckhoff_ER1xxx.Beckhoff_ER1xxxEK1122.A_0016_ER1819_0021_0017.Channel_12.Input <-> Channel 12/Input
//     PlcTask Inputs/GVL_iXlinker.EtherCAT_Master_ERxxxx.Beckhoff_ER1xxx.Beckhoff_ER1xxxEK1122.A_0016_ER1819_0021_0017.Channel_13.Input <-> Channel 13/Input
//     PlcTask Inputs/GVL_iXlinker.EtherCAT_Master_ERxxxx.Beckhoff_ER1xxx.Beckhoff_ER1xxxEK1122.A_0016_ER1819_0021_0017.Channel_14.Input <-> Channel 14/Input
//     PlcTask Inputs/GVL_iXlinker.EtherCAT_Master_ERxxxx.Beckhoff_ER1xxx.Beckhoff_ER1xxxEK1122.A_0016_ER1819_0021_0017.Channel_15.Input <-> Channel 15/Input
//     PlcTask Inputs/GVL_iXlinker.EtherCAT_Master_ERxxxx.Beckhoff_ER1xxx.Beckhoff_ER1xxxEK1122.A_0016_ER1819_0021_0017.Channel_16.Input <-> Channel 16/Input
//     PlcTask Inputs/GVL_iXlinker.EtherCAT_Master_ERxxxx.Beckhoff_ER1xxx.Beckhoff_ER1xxxEK1122.A_0016_ER1819_0021_0017.WcState.WcState <-> WcState/WcState
//     PlcTask Inputs/GVL_iXlinker.EtherCAT_Master_ERxxxx.Beckhoff_ER1xxx.Beckhoff_ER1xxxEK1122.A_0016_ER1819_0021_0017.WcState.InputToggle <-> WcState/InputToggle
//     PlcTask Inputs/GVL_iXlinker.EtherCAT_Master_ERxxxx.Beckhoff_ER1xxx.Beckhoff_ER1xxxEK1122.A_0016_ER1819_0021_0017.InfoData.State <-> InfoData/State
//   PLC/PLC Instance <-> EtherCAT Master ERxxxx/Beckhoff ER1xxx/Beckhoff ER1xxxEK1122/A_0017(ER1819-0022-0017)
//     PlcTask Inputs/GVL_iXlinker.EtherCAT_Master_ERxxxx.Beckhoff_ER1xxx.Beckhoff_ER1xxxEK1122.A_0017_ER1819_0022_0017.Channel_1.Input <-> Channel 1/Input
//     PlcTask Inputs/GVL_iXlinker.EtherCAT_Master_ERxxxx.Beckhoff_ER1xxx.Beckhoff_ER1xxxEK1122.A_0017_ER1819_0022_0017.Channel_2.Input <-> Channel 2/Input
//     PlcTask Inputs/GVL_iXlinker.EtherCAT_Master_ERxxxx.Beckhoff_ER1xxx.Beckhoff_ER1xxxEK1122.A_0017_ER1819_0022_0017.Channel_3.Input <-> Channel 3/Input
//     PlcTask Inputs/GVL_iXlinker.EtherCAT_Master_ERxxxx.Beckhoff_ER1xxx.Beckhoff_ER1xxxEK1122.A_0017_ER1819_0022_0017.Channel_4.Input <-> Channel 4/Input
//     PlcTask Inputs/GVL_iXlinker.EtherCAT_Master_ERxxxx.Beckhoff_ER1xxx.Beckhoff_ER1xxxEK1122.A_0017_ER1819_0022_0017.Channel_5.Input <-> Channel 5/Input
//     PlcTask Inputs/GVL_iXlinker.EtherCAT_Master_ERxxxx.Beckhoff_ER1xxx.Beckhoff_ER1xxxEK1122.A_0017_ER1819_0022_0017.Channel_6.Input <-> Channel 6/Input
//     PlcTask Inputs/GVL_iXlinker.EtherCAT_Master_ERxxxx.Beckhoff_ER1xxx.Beckhoff_ER1xxxEK1122.A_0017_ER1819_0022_0017.Channel_7.Input <-> Channel 7/Input
//     PlcTask Inputs/GVL_iXlinker.EtherCAT_Master_ERxxxx.Beckhoff_ER1xxx.Beckhoff_ER1xxxEK1122.A_0017_ER1819_0022_0017.Channel_8.Input <-> Channel 8/Input
//     PlcTask Inputs/GVL_iXlinker.EtherCAT_Master_ERxxxx.Beckhoff_ER1xxx.Beckhoff_ER1xxxEK1122.A_0017_ER1819_0022_0017.Channel_9.Input <-> Channel 9/Input
//     PlcTask Inputs/GVL_iXlinker.EtherCAT_Master_ERxxxx.Beckhoff_ER1xxx.Beckhoff_ER1xxxEK1122.A_0017_ER1819_0022_0017.Channel_10.Input <-> Channel 10/Input
//     PlcTask Inputs/GVL_iXlinker.EtherCAT_Master_ERxxxx.Beckhoff_ER1xxx.Beckhoff_ER1xxxEK1122.A_0017_ER1819_0022_0017.Channel_11.Input <-> Channel 11/Input
//     PlcTask Inputs/GVL_iXlinker.EtherCAT_Master_ERxxxx.Beckhoff_ER1xxx.Beckhoff_ER1xxxEK1122.A_0017_ER1819_0022_0017.Channel_12.Input <-> Channel 12/Input
//     PlcTask Inputs/GVL_iXlinker.EtherCAT_Master_ERxxxx.Beckhoff_ER1xxx.Beckhoff_ER1xxxEK1122.A_0017_ER1819_0022_0017.Channel_13.Input <-> Channel 13/Input
//     PlcTask Inputs/GVL_iXlinker.EtherCAT_Master_ERxxxx.Beckhoff_ER1xxx.Beckhoff_ER1xxxEK1122.A_0017_ER1819_0022_0017.Channel_14.Input <-> Channel 14/Input
//     PlcTask Inputs/GVL_iXlinker.EtherCAT_Master_ERxxxx.Beckhoff_ER1xxx.Beckhoff_ER1xxxEK1122.A_0017_ER1819_0022_0017.Channel_15.Input <-> Channel 15/Input
//     PlcTask Inputs/GVL_iXlinker.EtherCAT_Master_ERxxxx.Beckhoff_ER1xxx.Beckhoff_ER1xxxEK1122.A_0017_ER1819_0022_0017.Channel_16.Input <-> Channel 16/Input
//     PlcTask Inputs/GVL_iXlinker.EtherCAT_Master_ERxxxx.Beckhoff_ER1xxx.Beckhoff_ER1xxxEK1122.A_0017_ER1819_0022_0017.WcState.WcState <-> WcState/WcState
//     PlcTask Inputs/GVL_iXlinker.EtherCAT_Master_ERxxxx.Beckhoff_ER1xxx.Beckhoff_ER1xxxEK1122.A_0017_ER1819_0022_0017.WcState.InputToggle <-> WcState/InputToggle
//     PlcTask Inputs/GVL_iXlinker.EtherCAT_Master_ERxxxx.Beckhoff_ER1xxx.Beckhoff_ER1xxxEK1122.A_0017_ER1819_0022_0017.InfoData.State <-> InfoData/State
//   PLC/PLC Instance <-> EtherCAT Master ERxxxx/Beckhoff ER2xxx
//     PlcTask Inputs/GVL_iXlinker.EtherCAT_Master_ERxxxx.Beckhoff_ER2xxx.InfoData.State <-> InfoData/State
//   PLC/PLC Instance <-> EtherCAT Master ERxxxx/Beckhoff ER2xxx/Beckhoff ER2xxxEK1122
//     PlcTask Inputs/GVL_iXlinker.EtherCAT_Master_ERxxxx.Beckhoff_ER2xxx.Beckhoff_ER2xxxEK1122.InfoData.State <-> InfoData/State
//   PLC/PLC Instance <-> EtherCAT Master ERxxxx/Beckhoff ER2xxx/Beckhoff ER2xxxEK1122/Beckhoff ER2xxxsub EK1100
//     PlcTask Inputs/GVL_iXlinker.EtherCAT_Master_ERxxxx.Beckhoff_ER2xxx.Beckhoff_ER2xxxEK1122.Beckhoff_ER2xxxsub_EK1100.InfoData.State <-> InfoData/State
//   PLC/PLC Instance <-> EtherCAT Master ERxxxx/Beckhoff ER2xxx/Beckhoff ER2xxxEK1122/A_0001(ER2008-0001-0018)
//     PlcTask Outputs/GVL_iXlinker.EtherCAT_Master_ERxxxx.Beckhoff_ER2xxx.Beckhoff_ER2xxxEK1122.A_0001_ER2008_0001_0018.Channel_1.Output <-> Channel 1/Output
//     PlcTask Outputs/GVL_iXlinker.EtherCAT_Master_ERxxxx.Beckhoff_ER2xxx.Beckhoff_ER2xxxEK1122.A_0001_ER2008_0001_0018.Channel_2.Output <-> Channel 2/Output
//     PlcTask Outputs/GVL_iXlinker.EtherCAT_Master_ERxxxx.Beckhoff_ER2xxx.Beckhoff_ER2xxxEK1122.A_0001_ER2008_0001_0018.Channel_3.Output <-> Channel 3/Output
//     PlcTask Outputs/GVL_iXlinker.EtherCAT_Master_ERxxxx.Beckhoff_ER2xxx.Beckhoff_ER2xxxEK1122.A_0001_ER2008_0001_0018.Channel_4.Output <-> Channel 4/Output
//     PlcTask Outputs/GVL_iXlinker.EtherCAT_Master_ERxxxx.Beckhoff_ER2xxx.Beckhoff_ER2xxxEK1122.A_0001_ER2008_0001_0018.Channel_5.Output <-> Channel 5/Output
//     PlcTask Outputs/GVL_iXlinker.EtherCAT_Master_ERxxxx.Beckhoff_ER2xxx.Beckhoff_ER2xxxEK1122.A_0001_ER2008_0001_0018.Channel_6.Output <-> Channel 6/Output
//     PlcTask Outputs/GVL_iXlinker.EtherCAT_Master_ERxxxx.Beckhoff_ER2xxx.Beckhoff_ER2xxxEK1122.A_0001_ER2008_0001_0018.Channel_7.Output <-> Channel 7/Output
//     PlcTask Outputs/GVL_iXlinker.EtherCAT_Master_ERxxxx.Beckhoff_ER2xxx.Beckhoff_ER2xxxEK1122.A_0001_ER2008_0001_0018.Channel_8.Output <-> Channel 8/Output
//     PlcTask Inputs/GVL_iXlinker.EtherCAT_Master_ERxxxx.Beckhoff_ER2xxx.Beckhoff_ER2xxxEK1122.A_0001_ER2008_0001_0018.WcState.WcState <-> WcState/WcState
//     PlcTask Inputs/GVL_iXlinker.EtherCAT_Master_ERxxxx.Beckhoff_ER2xxx.Beckhoff_ER2xxxEK1122.A_0001_ER2008_0001_0018.InfoData.State <-> InfoData/State
//   PLC/PLC Instance <-> EtherCAT Master ERxxxx/Beckhoff ER2xxx/Beckhoff ER2xxxEK1122/A_0002(ER2008-0001-0019)
//     PlcTask Outputs/GVL_iXlinker.EtherCAT_Master_ERxxxx.Beckhoff_ER2xxx.Beckhoff_ER2xxxEK1122.A_0002_ER2008_0001_0019.Channel_1.Output <-> Channel 1/Output
//     PlcTask Outputs/GVL_iXlinker.EtherCAT_Master_ERxxxx.Beckhoff_ER2xxx.Beckhoff_ER2xxxEK1122.A_0002_ER2008_0001_0019.Channel_2.Output <-> Channel 2/Output
//     PlcTask Outputs/GVL_iXlinker.EtherCAT_Master_ERxxxx.Beckhoff_ER2xxx.Beckhoff_ER2xxxEK1122.A_0002_ER2008_0001_0019.Channel_3.Output <-> Channel 3/Output
//     PlcTask Outputs/GVL_iXlinker.EtherCAT_Master_ERxxxx.Beckhoff_ER2xxx.Beckhoff_ER2xxxEK1122.A_0002_ER2008_0001_0019.Channel_4.Output <-> Channel 4/Output
//     PlcTask Outputs/GVL_iXlinker.EtherCAT_Master_ERxxxx.Beckhoff_ER2xxx.Beckhoff_ER2xxxEK1122.A_0002_ER2008_0001_0019.Channel_5.Output <-> Channel 5/Output
//     PlcTask Outputs/GVL_iXlinker.EtherCAT_Master_ERxxxx.Beckhoff_ER2xxx.Beckhoff_ER2xxxEK1122.A_0002_ER2008_0001_0019.Channel_6.Output <-> Channel 6/Output
//     PlcTask Outputs/GVL_iXlinker.EtherCAT_Master_ERxxxx.Beckhoff_ER2xxx.Beckhoff_ER2xxxEK1122.A_0002_ER2008_0001_0019.Channel_7.Output <-> Channel 7/Output
//     PlcTask Outputs/GVL_iXlinker.EtherCAT_Master_ERxxxx.Beckhoff_ER2xxx.Beckhoff_ER2xxxEK1122.A_0002_ER2008_0001_0019.Channel_8.Output <-> Channel 8/Output
//     PlcTask Inputs/GVL_iXlinker.EtherCAT_Master_ERxxxx.Beckhoff_ER2xxx.Beckhoff_ER2xxxEK1122.A_0002_ER2008_0001_0019.WcState.WcState <-> WcState/WcState
//     PlcTask Inputs/GVL_iXlinker.EtherCAT_Master_ERxxxx.Beckhoff_ER2xxx.Beckhoff_ER2xxxEK1122.A_0002_ER2008_0001_0019.InfoData.State <-> InfoData/State
//   PLC/PLC Instance <-> EtherCAT Master ERxxxx/Beckhoff ER2xxx/Beckhoff ER2xxxEK1122/A_0003(ER2008-0002-0018)
//     PlcTask Outputs/GVL_iXlinker.EtherCAT_Master_ERxxxx.Beckhoff_ER2xxx.Beckhoff_ER2xxxEK1122.A_0003_ER2008_0002_0018.Channel_1.Output <-> Channel 1/Output
//     PlcTask Outputs/GVL_iXlinker.EtherCAT_Master_ERxxxx.Beckhoff_ER2xxx.Beckhoff_ER2xxxEK1122.A_0003_ER2008_0002_0018.Channel_2.Output <-> Channel 2/Output
//     PlcTask Outputs/GVL_iXlinker.EtherCAT_Master_ERxxxx.Beckhoff_ER2xxx.Beckhoff_ER2xxxEK1122.A_0003_ER2008_0002_0018.Channel_3.Output <-> Channel 3/Output
//     PlcTask Outputs/GVL_iXlinker.EtherCAT_Master_ERxxxx.Beckhoff_ER2xxx.Beckhoff_ER2xxxEK1122.A_0003_ER2008_0002_0018.Channel_4.Output <-> Channel 4/Output
//     PlcTask Outputs/GVL_iXlinker.EtherCAT_Master_ERxxxx.Beckhoff_ER2xxx.Beckhoff_ER2xxxEK1122.A_0003_ER2008_0002_0018.Channel_5.Output <-> Channel 5/Output
//     PlcTask Outputs/GVL_iXlinker.EtherCAT_Master_ERxxxx.Beckhoff_ER2xxx.Beckhoff_ER2xxxEK1122.A_0003_ER2008_0002_0018.Channel_6.Output <-> Channel 6/Output
//     PlcTask Outputs/GVL_iXlinker.EtherCAT_Master_ERxxxx.Beckhoff_ER2xxx.Beckhoff_ER2xxxEK1122.A_0003_ER2008_0002_0018.Channel_7.Output <-> Channel 7/Output
//     PlcTask Outputs/GVL_iXlinker.EtherCAT_Master_ERxxxx.Beckhoff_ER2xxx.Beckhoff_ER2xxxEK1122.A_0003_ER2008_0002_0018.Channel_8.Output <-> Channel 8/Output
//     PlcTask Inputs/GVL_iXlinker.EtherCAT_Master_ERxxxx.Beckhoff_ER2xxx.Beckhoff_ER2xxxEK1122.A_0003_ER2008_0002_0018.WcState.WcState <-> WcState/WcState
//     PlcTask Inputs/GVL_iXlinker.EtherCAT_Master_ERxxxx.Beckhoff_ER2xxx.Beckhoff_ER2xxxEK1122.A_0003_ER2008_0002_0018.InfoData.State <-> InfoData/State
//   PLC/PLC Instance <-> EtherCAT Master ERxxxx/Beckhoff ER2xxx/Beckhoff ER2xxxEK1122/A_0004(ER2008-0002-0019)
//     PlcTask Outputs/GVL_iXlinker.EtherCAT_Master_ERxxxx.Beckhoff_ER2xxx.Beckhoff_ER2xxxEK1122.A_0004_ER2008_0002_0019.Channel_1.Output <-> Channel 1/Output
//     PlcTask Outputs/GVL_iXlinker.EtherCAT_Master_ERxxxx.Beckhoff_ER2xxx.Beckhoff_ER2xxxEK1122.A_0004_ER2008_0002_0019.Channel_2.Output <-> Channel 2/Output
//     PlcTask Outputs/GVL_iXlinker.EtherCAT_Master_ERxxxx.Beckhoff_ER2xxx.Beckhoff_ER2xxxEK1122.A_0004_ER2008_0002_0019.Channel_3.Output <-> Channel 3/Output
//     PlcTask Outputs/GVL_iXlinker.EtherCAT_Master_ERxxxx.Beckhoff_ER2xxx.Beckhoff_ER2xxxEK1122.A_0004_ER2008_0002_0019.Channel_4.Output <-> Channel 4/Output
//     PlcTask Outputs/GVL_iXlinker.EtherCAT_Master_ERxxxx.Beckhoff_ER2xxx.Beckhoff_ER2xxxEK1122.A_0004_ER2008_0002_0019.Channel_5.Output <-> Channel 5/Output
//     PlcTask Outputs/GVL_iXlinker.EtherCAT_Master_ERxxxx.Beckhoff_ER2xxx.Beckhoff_ER2xxxEK1122.A_0004_ER2008_0002_0019.Channel_6.Output <-> Channel 6/Output
//     PlcTask Outputs/GVL_iXlinker.EtherCAT_Master_ERxxxx.Beckhoff_ER2xxx.Beckhoff_ER2xxxEK1122.A_0004_ER2008_0002_0019.Channel_7.Output <-> Channel 7/Output
//     PlcTask Outputs/GVL_iXlinker.EtherCAT_Master_ERxxxx.Beckhoff_ER2xxx.Beckhoff_ER2xxxEK1122.A_0004_ER2008_0002_0019.Channel_8.Output <-> Channel 8/Output
//     PlcTask Inputs/GVL_iXlinker.EtherCAT_Master_ERxxxx.Beckhoff_ER2xxx.Beckhoff_ER2xxxEK1122.A_0004_ER2008_0002_0019.WcState.WcState <-> WcState/WcState
//     PlcTask Inputs/GVL_iXlinker.EtherCAT_Master_ERxxxx.Beckhoff_ER2xxx.Beckhoff_ER2xxxEK1122.A_0004_ER2008_0002_0019.InfoData.State <-> InfoData/State
//   PLC/PLC Instance <-> EtherCAT Master ERxxxx/Beckhoff ER2xxx/Beckhoff ER2xxxEK1122/A_0005(ER2008-0022-0017)
//     PlcTask Outputs/GVL_iXlinker.EtherCAT_Master_ERxxxx.Beckhoff_ER2xxx.Beckhoff_ER2xxxEK1122.A_0005_ER2008_0022_0017.Channel_1.Output <-> Channel 1/Output
//     PlcTask Outputs/GVL_iXlinker.EtherCAT_Master_ERxxxx.Beckhoff_ER2xxx.Beckhoff_ER2xxxEK1122.A_0005_ER2008_0022_0017.Channel_2.Output <-> Channel 2/Output
//     PlcTask Outputs/GVL_iXlinker.EtherCAT_Master_ERxxxx.Beckhoff_ER2xxx.Beckhoff_ER2xxxEK1122.A_0005_ER2008_0022_0017.Channel_3.Output <-> Channel 3/Output
//     PlcTask Outputs/GVL_iXlinker.EtherCAT_Master_ERxxxx.Beckhoff_ER2xxx.Beckhoff_ER2xxxEK1122.A_0005_ER2008_0022_0017.Channel_4.Output <-> Channel 4/Output
//     PlcTask Outputs/GVL_iXlinker.EtherCAT_Master_ERxxxx.Beckhoff_ER2xxx.Beckhoff_ER2xxxEK1122.A_0005_ER2008_0022_0017.Channel_5.Output <-> Channel 5/Output
//     PlcTask Outputs/GVL_iXlinker.EtherCAT_Master_ERxxxx.Beckhoff_ER2xxx.Beckhoff_ER2xxxEK1122.A_0005_ER2008_0022_0017.Channel_6.Output <-> Channel 6/Output
//     PlcTask Outputs/GVL_iXlinker.EtherCAT_Master_ERxxxx.Beckhoff_ER2xxx.Beckhoff_ER2xxxEK1122.A_0005_ER2008_0022_0017.Channel_7.Output <-> Channel 7/Output
//     PlcTask Outputs/GVL_iXlinker.EtherCAT_Master_ERxxxx.Beckhoff_ER2xxx.Beckhoff_ER2xxxEK1122.A_0005_ER2008_0022_0017.Channel_8.Output <-> Channel 8/Output
//     PlcTask Inputs/GVL_iXlinker.EtherCAT_Master_ERxxxx.Beckhoff_ER2xxx.Beckhoff_ER2xxxEK1122.A_0005_ER2008_0022_0017.WcState.WcState <-> WcState/WcState
//     PlcTask Inputs/GVL_iXlinker.EtherCAT_Master_ERxxxx.Beckhoff_ER2xxx.Beckhoff_ER2xxxEK1122.A_0005_ER2008_0022_0017.InfoData.State <-> InfoData/State
//   PLC/PLC Instance <-> EtherCAT Master ERxxxx/Beckhoff ER2xxx/Beckhoff ER2xxxEK1122/A_0006(ER2008-0022-0018)
//     PlcTask Outputs/GVL_iXlinker.EtherCAT_Master_ERxxxx.Beckhoff_ER2xxx.Beckhoff_ER2xxxEK1122.A_0006_ER2008_0022_0018.Channel_1.Output <-> Channel 1/Output
//     PlcTask Outputs/GVL_iXlinker.EtherCAT_Master_ERxxxx.Beckhoff_ER2xxx.Beckhoff_ER2xxxEK1122.A_0006_ER2008_0022_0018.Channel_2.Output <-> Channel 2/Output
//     PlcTask Outputs/GVL_iXlinker.EtherCAT_Master_ERxxxx.Beckhoff_ER2xxx.Beckhoff_ER2xxxEK1122.A_0006_ER2008_0022_0018.Channel_3.Output <-> Channel 3/Output
//     PlcTask Outputs/GVL_iXlinker.EtherCAT_Master_ERxxxx.Beckhoff_ER2xxx.Beckhoff_ER2xxxEK1122.A_0006_ER2008_0022_0018.Channel_4.Output <-> Channel 4/Output
//     PlcTask Outputs/GVL_iXlinker.EtherCAT_Master_ERxxxx.Beckhoff_ER2xxx.Beckhoff_ER2xxxEK1122.A_0006_ER2008_0022_0018.Channel_5.Output <-> Channel 5/Output
//     PlcTask Outputs/GVL_iXlinker.EtherCAT_Master_ERxxxx.Beckhoff_ER2xxx.Beckhoff_ER2xxxEK1122.A_0006_ER2008_0022_0018.Channel_6.Output <-> Channel 6/Output
//     PlcTask Outputs/GVL_iXlinker.EtherCAT_Master_ERxxxx.Beckhoff_ER2xxx.Beckhoff_ER2xxxEK1122.A_0006_ER2008_0022_0018.Channel_7.Output <-> Channel 7/Output
//     PlcTask Outputs/GVL_iXlinker.EtherCAT_Master_ERxxxx.Beckhoff_ER2xxx.Beckhoff_ER2xxxEK1122.A_0006_ER2008_0022_0018.Channel_8.Output <-> Channel 8/Output
//     PlcTask Inputs/GVL_iXlinker.EtherCAT_Master_ERxxxx.Beckhoff_ER2xxx.Beckhoff_ER2xxxEK1122.A_0006_ER2008_0022_0018.WcState.WcState <-> WcState/WcState
//     PlcTask Inputs/GVL_iXlinker.EtherCAT_Master_ERxxxx.Beckhoff_ER2xxx.Beckhoff_ER2xxxEK1122.A_0006_ER2008_0022_0018.InfoData.State <-> InfoData/State
//   PLC/PLC Instance <-> EtherCAT Master ERxxxx/Beckhoff ER2xxx/Beckhoff ER2xxxEK1122/A_0007(ER2028-0001-0017)
//     PlcTask Outputs/GVL_iXlinker.EtherCAT_Master_ERxxxx.Beckhoff_ER2xxx.Beckhoff_ER2xxxEK1122.A_0007_ER2028_0001_0017.Channel_1.Output <-> Channel 1/Output
//     PlcTask Outputs/GVL_iXlinker.EtherCAT_Master_ERxxxx.Beckhoff_ER2xxx.Beckhoff_ER2xxxEK1122.A_0007_ER2028_0001_0017.Channel_2.Output <-> Channel 2/Output
//     PlcTask Outputs/GVL_iXlinker.EtherCAT_Master_ERxxxx.Beckhoff_ER2xxx.Beckhoff_ER2xxxEK1122.A_0007_ER2028_0001_0017.Channel_3.Output <-> Channel 3/Output
//     PlcTask Outputs/GVL_iXlinker.EtherCAT_Master_ERxxxx.Beckhoff_ER2xxx.Beckhoff_ER2xxxEK1122.A_0007_ER2028_0001_0017.Channel_4.Output <-> Channel 4/Output
//     PlcTask Outputs/GVL_iXlinker.EtherCAT_Master_ERxxxx.Beckhoff_ER2xxx.Beckhoff_ER2xxxEK1122.A_0007_ER2028_0001_0017.Channel_5.Output <-> Channel 5/Output
//     PlcTask Outputs/GVL_iXlinker.EtherCAT_Master_ERxxxx.Beckhoff_ER2xxx.Beckhoff_ER2xxxEK1122.A_0007_ER2028_0001_0017.Channel_6.Output <-> Channel 6/Output
//     PlcTask Outputs/GVL_iXlinker.EtherCAT_Master_ERxxxx.Beckhoff_ER2xxx.Beckhoff_ER2xxxEK1122.A_0007_ER2028_0001_0017.Channel_7.Output <-> Channel 7/Output
//     PlcTask Outputs/GVL_iXlinker.EtherCAT_Master_ERxxxx.Beckhoff_ER2xxx.Beckhoff_ER2xxxEK1122.A_0007_ER2028_0001_0017.Channel_8.Output <-> Channel 8/Output
//     PlcTask Inputs/GVL_iXlinker.EtherCAT_Master_ERxxxx.Beckhoff_ER2xxx.Beckhoff_ER2xxxEK1122.A_0007_ER2028_0001_0017.WcState.WcState <-> WcState/WcState
//     PlcTask Inputs/GVL_iXlinker.EtherCAT_Master_ERxxxx.Beckhoff_ER2xxx.Beckhoff_ER2xxxEK1122.A_0007_ER2028_0001_0017.InfoData.State <-> InfoData/State
//   PLC/PLC Instance <-> EtherCAT Master ERxxxx/Beckhoff ER2xxx/Beckhoff ER2xxxEK1122/A_0008(ER2028-0001-0018)
//     PlcTask Outputs/GVL_iXlinker.EtherCAT_Master_ERxxxx.Beckhoff_ER2xxx.Beckhoff_ER2xxxEK1122.A_0008_ER2028_0001_0018.Channel_1.Output <-> Channel 1/Output
//     PlcTask Outputs/GVL_iXlinker.EtherCAT_Master_ERxxxx.Beckhoff_ER2xxx.Beckhoff_ER2xxxEK1122.A_0008_ER2028_0001_0018.Channel_2.Output <-> Channel 2/Output
//     PlcTask Outputs/GVL_iXlinker.EtherCAT_Master_ERxxxx.Beckhoff_ER2xxx.Beckhoff_ER2xxxEK1122.A_0008_ER2028_0001_0018.Channel_3.Output <-> Channel 3/Output
//     PlcTask Outputs/GVL_iXlinker.EtherCAT_Master_ERxxxx.Beckhoff_ER2xxx.Beckhoff_ER2xxxEK1122.A_0008_ER2028_0001_0018.Channel_4.Output <-> Channel 4/Output
//     PlcTask Outputs/GVL_iXlinker.EtherCAT_Master_ERxxxx.Beckhoff_ER2xxx.Beckhoff_ER2xxxEK1122.A_0008_ER2028_0001_0018.Channel_5.Output <-> Channel 5/Output
//     PlcTask Outputs/GVL_iXlinker.EtherCAT_Master_ERxxxx.Beckhoff_ER2xxx.Beckhoff_ER2xxxEK1122.A_0008_ER2028_0001_0018.Channel_6.Output <-> Channel 6/Output
//     PlcTask Outputs/GVL_iXlinker.EtherCAT_Master_ERxxxx.Beckhoff_ER2xxx.Beckhoff_ER2xxxEK1122.A_0008_ER2028_0001_0018.Channel_7.Output <-> Channel 7/Output
//     PlcTask Outputs/GVL_iXlinker.EtherCAT_Master_ERxxxx.Beckhoff_ER2xxx.Beckhoff_ER2xxxEK1122.A_0008_ER2028_0001_0018.Channel_8.Output <-> Channel 8/Output
//     PlcTask Inputs/GVL_iXlinker.EtherCAT_Master_ERxxxx.Beckhoff_ER2xxx.Beckhoff_ER2xxxEK1122.A_0008_ER2028_0001_0018.WcState.WcState <-> WcState/WcState
//     PlcTask Inputs/GVL_iXlinker.EtherCAT_Master_ERxxxx.Beckhoff_ER2xxx.Beckhoff_ER2xxxEK1122.A_0008_ER2028_0001_0018.InfoData.State <-> InfoData/State
//   PLC/PLC Instance <-> EtherCAT Master ERxxxx/Beckhoff ER2xxx/Beckhoff ER2xxxEK1122/A_0009(ER2028-0002-0018)
//     PlcTask Outputs/GVL_iXlinker.EtherCAT_Master_ERxxxx.Beckhoff_ER2xxx.Beckhoff_ER2xxxEK1122.A_0009_ER2028_0002_0018.Channel_1.Output <-> Channel 1/Output
//     PlcTask Outputs/GVL_iXlinker.EtherCAT_Master_ERxxxx.Beckhoff_ER2xxx.Beckhoff_ER2xxxEK1122.A_0009_ER2028_0002_0018.Channel_2.Output <-> Channel 2/Output
//     PlcTask Outputs/GVL_iXlinker.EtherCAT_Master_ERxxxx.Beckhoff_ER2xxx.Beckhoff_ER2xxxEK1122.A_0009_ER2028_0002_0018.Channel_3.Output <-> Channel 3/Output
//     PlcTask Outputs/GVL_iXlinker.EtherCAT_Master_ERxxxx.Beckhoff_ER2xxx.Beckhoff_ER2xxxEK1122.A_0009_ER2028_0002_0018.Channel_4.Output <-> Channel 4/Output
//     PlcTask Outputs/GVL_iXlinker.EtherCAT_Master_ERxxxx.Beckhoff_ER2xxx.Beckhoff_ER2xxxEK1122.A_0009_ER2028_0002_0018.Channel_5.Output <-> Channel 5/Output
//     PlcTask Outputs/GVL_iXlinker.EtherCAT_Master_ERxxxx.Beckhoff_ER2xxx.Beckhoff_ER2xxxEK1122.A_0009_ER2028_0002_0018.Channel_6.Output <-> Channel 6/Output
//     PlcTask Outputs/GVL_iXlinker.EtherCAT_Master_ERxxxx.Beckhoff_ER2xxx.Beckhoff_ER2xxxEK1122.A_0009_ER2028_0002_0018.Channel_7.Output <-> Channel 7/Output
//     PlcTask Outputs/GVL_iXlinker.EtherCAT_Master_ERxxxx.Beckhoff_ER2xxx.Beckhoff_ER2xxxEK1122.A_0009_ER2028_0002_0018.Channel_8.Output <-> Channel 8/Output
//     PlcTask Inputs/GVL_iXlinker.EtherCAT_Master_ERxxxx.Beckhoff_ER2xxx.Beckhoff_ER2xxxEK1122.A_0009_ER2028_0002_0018.WcState.WcState <-> WcState/WcState
//     PlcTask Inputs/GVL_iXlinker.EtherCAT_Master_ERxxxx.Beckhoff_ER2xxx.Beckhoff_ER2xxxEK1122.A_0009_ER2028_0002_0018.InfoData.State <-> InfoData/State
//   PLC/PLC Instance <-> EtherCAT Master ERxxxx/Beckhoff ER2xxx/Beckhoff ER2xxxEK1122/A_0010(ER2028-0002-0019)
//     PlcTask Outputs/GVL_iXlinker.EtherCAT_Master_ERxxxx.Beckhoff_ER2xxx.Beckhoff_ER2xxxEK1122.A_0010_ER2028_0002_0019.Channel_1.Output <-> Channel 1/Output
//     PlcTask Outputs/GVL_iXlinker.EtherCAT_Master_ERxxxx.Beckhoff_ER2xxx.Beckhoff_ER2xxxEK1122.A_0010_ER2028_0002_0019.Channel_2.Output <-> Channel 2/Output
//     PlcTask Outputs/GVL_iXlinker.EtherCAT_Master_ERxxxx.Beckhoff_ER2xxx.Beckhoff_ER2xxxEK1122.A_0010_ER2028_0002_0019.Channel_3.Output <-> Channel 3/Output
//     PlcTask Outputs/GVL_iXlinker.EtherCAT_Master_ERxxxx.Beckhoff_ER2xxx.Beckhoff_ER2xxxEK1122.A_0010_ER2028_0002_0019.Channel_4.Output <-> Channel 4/Output
//     PlcTask Outputs/GVL_iXlinker.EtherCAT_Master_ERxxxx.Beckhoff_ER2xxx.Beckhoff_ER2xxxEK1122.A_0010_ER2028_0002_0019.Channel_5.Output <-> Channel 5/Output
//     PlcTask Outputs/GVL_iXlinker.EtherCAT_Master_ERxxxx.Beckhoff_ER2xxx.Beckhoff_ER2xxxEK1122.A_0010_ER2028_0002_0019.Channel_6.Output <-> Channel 6/Output
//     PlcTask Outputs/GVL_iXlinker.EtherCAT_Master_ERxxxx.Beckhoff_ER2xxx.Beckhoff_ER2xxxEK1122.A_0010_ER2028_0002_0019.Channel_7.Output <-> Channel 7/Output
//     PlcTask Outputs/GVL_iXlinker.EtherCAT_Master_ERxxxx.Beckhoff_ER2xxx.Beckhoff_ER2xxxEK1122.A_0010_ER2028_0002_0019.Channel_8.Output <-> Channel 8/Output
//     PlcTask Inputs/GVL_iXlinker.EtherCAT_Master_ERxxxx.Beckhoff_ER2xxx.Beckhoff_ER2xxxEK1122.A_0010_ER2028_0002_0019.WcState.WcState <-> WcState/WcState
//     PlcTask Inputs/GVL_iXlinker.EtherCAT_Master_ERxxxx.Beckhoff_ER2xxx.Beckhoff_ER2xxxEK1122.A_0010_ER2028_0002_0019.InfoData.State <-> InfoData/State
//   PLC/PLC Instance <-> EtherCAT Master ERxxxx/Beckhoff ER2xxx/Beckhoff ER2xxxEK1122/A_0011(ER2028-1032-0016)
//     PlcTask Outputs/GVL_iXlinker.EtherCAT_Master_ERxxxx.Beckhoff_ER2xxx.Beckhoff_ER2xxxEK1122.A_0011_ER2028_1032_0016.Channel_1.Output <-> Channel 1/Output
//     PlcTask Outputs/GVL_iXlinker.EtherCAT_Master_ERxxxx.Beckhoff_ER2xxx.Beckhoff_ER2xxxEK1122.A_0011_ER2028_1032_0016.Channel_2.Output <-> Channel 2/Output
//     PlcTask Outputs/GVL_iXlinker.EtherCAT_Master_ERxxxx.Beckhoff_ER2xxx.Beckhoff_ER2xxxEK1122.A_0011_ER2028_1032_0016.Channel_3.Output <-> Channel 3/Output
//     PlcTask Outputs/GVL_iXlinker.EtherCAT_Master_ERxxxx.Beckhoff_ER2xxx.Beckhoff_ER2xxxEK1122.A_0011_ER2028_1032_0016.Channel_4.Output <-> Channel 4/Output
//     PlcTask Outputs/GVL_iXlinker.EtherCAT_Master_ERxxxx.Beckhoff_ER2xxx.Beckhoff_ER2xxxEK1122.A_0011_ER2028_1032_0016.Channel_5.Output <-> Channel 5/Output
//     PlcTask Outputs/GVL_iXlinker.EtherCAT_Master_ERxxxx.Beckhoff_ER2xxx.Beckhoff_ER2xxxEK1122.A_0011_ER2028_1032_0016.Channel_6.Output <-> Channel 6/Output
//     PlcTask Outputs/GVL_iXlinker.EtherCAT_Master_ERxxxx.Beckhoff_ER2xxx.Beckhoff_ER2xxxEK1122.A_0011_ER2028_1032_0016.Channel_7.Output <-> Channel 7/Output
//     PlcTask Outputs/GVL_iXlinker.EtherCAT_Master_ERxxxx.Beckhoff_ER2xxx.Beckhoff_ER2xxxEK1122.A_0011_ER2028_1032_0016.Channel_8.Output <-> Channel 8/Output
//     PlcTask Inputs/GVL_iXlinker.EtherCAT_Master_ERxxxx.Beckhoff_ER2xxx.Beckhoff_ER2xxxEK1122.A_0011_ER2028_1032_0016.WcState.WcState <-> WcState/WcState
//     PlcTask Inputs/GVL_iXlinker.EtherCAT_Master_ERxxxx.Beckhoff_ER2xxx.Beckhoff_ER2xxxEK1122.A_0011_ER2028_1032_0016.InfoData.State <-> InfoData/State
//   PLC/PLC Instance <-> EtherCAT Master ERxxxx/Beckhoff ER2xxx/Beckhoff ER2xxxEK1122/A_0012(ER2038-0001-0017)
//     PlcTask Inputs/GVL_iXlinker.EtherCAT_Master_ERxxxx.Beckhoff_ER2xxx.Beckhoff_ER2xxxEK1122.A_0012_ER2038_0001_0017.Diag_Channel_1.Input <-> Diag Channel 1/Input
//     PlcTask Inputs/GVL_iXlinker.EtherCAT_Master_ERxxxx.Beckhoff_ER2xxx.Beckhoff_ER2xxxEK1122.A_0012_ER2038_0001_0017.Diag_Channel_2.Input <-> Diag Channel 2/Input
//     PlcTask Inputs/GVL_iXlinker.EtherCAT_Master_ERxxxx.Beckhoff_ER2xxx.Beckhoff_ER2xxxEK1122.A_0012_ER2038_0001_0017.Diag_Channel_3.Input <-> Diag Channel 3/Input
//     PlcTask Inputs/GVL_iXlinker.EtherCAT_Master_ERxxxx.Beckhoff_ER2xxx.Beckhoff_ER2xxxEK1122.A_0012_ER2038_0001_0017.Diag_Channel_4.Input <-> Diag Channel 4/Input
//     PlcTask Inputs/GVL_iXlinker.EtherCAT_Master_ERxxxx.Beckhoff_ER2xxx.Beckhoff_ER2xxxEK1122.A_0012_ER2038_0001_0017.Diag_Channel_5.Input <-> Diag Channel 5/Input
//     PlcTask Inputs/GVL_iXlinker.EtherCAT_Master_ERxxxx.Beckhoff_ER2xxx.Beckhoff_ER2xxxEK1122.A_0012_ER2038_0001_0017.Diag_Channel_6.Input <-> Diag Channel 6/Input
//     PlcTask Inputs/GVL_iXlinker.EtherCAT_Master_ERxxxx.Beckhoff_ER2xxx.Beckhoff_ER2xxxEK1122.A_0012_ER2038_0001_0017.Diag_Channel_7.Input <-> Diag Channel 7/Input
//     PlcTask Inputs/GVL_iXlinker.EtherCAT_Master_ERxxxx.Beckhoff_ER2xxx.Beckhoff_ER2xxxEK1122.A_0012_ER2038_0001_0017.Diag_Channel_8.Input <-> Diag Channel 8/Input
//     PlcTask Outputs/GVL_iXlinker.EtherCAT_Master_ERxxxx.Beckhoff_ER2xxx.Beckhoff_ER2xxxEK1122.A_0012_ER2038_0001_0017.Channel_1.Output <-> Channel 1/Output
//     PlcTask Outputs/GVL_iXlinker.EtherCAT_Master_ERxxxx.Beckhoff_ER2xxx.Beckhoff_ER2xxxEK1122.A_0012_ER2038_0001_0017.Channel_2.Output <-> Channel 2/Output
//     PlcTask Outputs/GVL_iXlinker.EtherCAT_Master_ERxxxx.Beckhoff_ER2xxx.Beckhoff_ER2xxxEK1122.A_0012_ER2038_0001_0017.Channel_3.Output <-> Channel 3/Output
//     PlcTask Outputs/GVL_iXlinker.EtherCAT_Master_ERxxxx.Beckhoff_ER2xxx.Beckhoff_ER2xxxEK1122.A_0012_ER2038_0001_0017.Channel_4.Output <-> Channel 4/Output
//     PlcTask Outputs/GVL_iXlinker.EtherCAT_Master_ERxxxx.Beckhoff_ER2xxx.Beckhoff_ER2xxxEK1122.A_0012_ER2038_0001_0017.Channel_5.Output <-> Channel 5/Output
//     PlcTask Outputs/GVL_iXlinker.EtherCAT_Master_ERxxxx.Beckhoff_ER2xxx.Beckhoff_ER2xxxEK1122.A_0012_ER2038_0001_0017.Channel_6.Output <-> Channel 6/Output
//     PlcTask Outputs/GVL_iXlinker.EtherCAT_Master_ERxxxx.Beckhoff_ER2xxx.Beckhoff_ER2xxxEK1122.A_0012_ER2038_0001_0017.Channel_7.Output <-> Channel 7/Output
//     PlcTask Outputs/GVL_iXlinker.EtherCAT_Master_ERxxxx.Beckhoff_ER2xxx.Beckhoff_ER2xxxEK1122.A_0012_ER2038_0001_0017.Channel_8.Output <-> Channel 8/Output
//     PlcTask Inputs/GVL_iXlinker.EtherCAT_Master_ERxxxx.Beckhoff_ER2xxx.Beckhoff_ER2xxxEK1122.A_0012_ER2038_0001_0017.WcState.WcState <-> WcState/WcState
//     PlcTask Inputs/GVL_iXlinker.EtherCAT_Master_ERxxxx.Beckhoff_ER2xxx.Beckhoff_ER2xxxEK1122.A_0012_ER2038_0001_0017.WcState.InputToggle <-> WcState/InputToggle
//     PlcTask Inputs/GVL_iXlinker.EtherCAT_Master_ERxxxx.Beckhoff_ER2xxx.Beckhoff_ER2xxxEK1122.A_0012_ER2038_0001_0017.InfoData.State <-> InfoData/State
//   PLC/PLC Instance <-> EtherCAT Master ERxxxx/Beckhoff ER2xxx/Beckhoff ER2xxxEK1122/A_0013(ER2038-0001-0018)
//     PlcTask Inputs/GVL_iXlinker.EtherCAT_Master_ERxxxx.Beckhoff_ER2xxx.Beckhoff_ER2xxxEK1122.A_0013_ER2038_0001_0018.Diag_Channel_1.Input <-> Diag Channel 1/Input
//     PlcTask Inputs/GVL_iXlinker.EtherCAT_Master_ERxxxx.Beckhoff_ER2xxx.Beckhoff_ER2xxxEK1122.A_0013_ER2038_0001_0018.Diag_Channel_2.Input <-> Diag Channel 2/Input
//     PlcTask Inputs/GVL_iXlinker.EtherCAT_Master_ERxxxx.Beckhoff_ER2xxx.Beckhoff_ER2xxxEK1122.A_0013_ER2038_0001_0018.Diag_Channel_3.Input <-> Diag Channel 3/Input
//     PlcTask Inputs/GVL_iXlinker.EtherCAT_Master_ERxxxx.Beckhoff_ER2xxx.Beckhoff_ER2xxxEK1122.A_0013_ER2038_0001_0018.Diag_Channel_4.Input <-> Diag Channel 4/Input
//     PlcTask Inputs/GVL_iXlinker.EtherCAT_Master_ERxxxx.Beckhoff_ER2xxx.Beckhoff_ER2xxxEK1122.A_0013_ER2038_0001_0018.Diag_Channel_5.Input <-> Diag Channel 5/Input
//     PlcTask Inputs/GVL_iXlinker.EtherCAT_Master_ERxxxx.Beckhoff_ER2xxx.Beckhoff_ER2xxxEK1122.A_0013_ER2038_0001_0018.Diag_Channel_6.Input <-> Diag Channel 6/Input
//     PlcTask Inputs/GVL_iXlinker.EtherCAT_Master_ERxxxx.Beckhoff_ER2xxx.Beckhoff_ER2xxxEK1122.A_0013_ER2038_0001_0018.Diag_Channel_7.Input <-> Diag Channel 7/Input
//     PlcTask Inputs/GVL_iXlinker.EtherCAT_Master_ERxxxx.Beckhoff_ER2xxx.Beckhoff_ER2xxxEK1122.A_0013_ER2038_0001_0018.Diag_Channel_8.Input <-> Diag Channel 8/Input
//     PlcTask Outputs/GVL_iXlinker.EtherCAT_Master_ERxxxx.Beckhoff_ER2xxx.Beckhoff_ER2xxxEK1122.A_0013_ER2038_0001_0018.Channel_1.Output <-> Channel 1/Output
//     PlcTask Outputs/GVL_iXlinker.EtherCAT_Master_ERxxxx.Beckhoff_ER2xxx.Beckhoff_ER2xxxEK1122.A_0013_ER2038_0001_0018.Channel_2.Output <-> Channel 2/Output
//     PlcTask Outputs/GVL_iXlinker.EtherCAT_Master_ERxxxx.Beckhoff_ER2xxx.Beckhoff_ER2xxxEK1122.A_0013_ER2038_0001_0018.Channel_3.Output <-> Channel 3/Output
//     PlcTask Outputs/GVL_iXlinker.EtherCAT_Master_ERxxxx.Beckhoff_ER2xxx.Beckhoff_ER2xxxEK1122.A_0013_ER2038_0001_0018.Channel_4.Output <-> Channel 4/Output
//     PlcTask Outputs/GVL_iXlinker.EtherCAT_Master_ERxxxx.Beckhoff_ER2xxx.Beckhoff_ER2xxxEK1122.A_0013_ER2038_0001_0018.Channel_5.Output <-> Channel 5/Output
//     PlcTask Outputs/GVL_iXlinker.EtherCAT_Master_ERxxxx.Beckhoff_ER2xxx.Beckhoff_ER2xxxEK1122.A_0013_ER2038_0001_0018.Channel_6.Output <-> Channel 6/Output
//     PlcTask Outputs/GVL_iXlinker.EtherCAT_Master_ERxxxx.Beckhoff_ER2xxx.Beckhoff_ER2xxxEK1122.A_0013_ER2038_0001_0018.Channel_7.Output <-> Channel 7/Output
//     PlcTask Outputs/GVL_iXlinker.EtherCAT_Master_ERxxxx.Beckhoff_ER2xxx.Beckhoff_ER2xxxEK1122.A_0013_ER2038_0001_0018.Channel_8.Output <-> Channel 8/Output
//     PlcTask Inputs/GVL_iXlinker.EtherCAT_Master_ERxxxx.Beckhoff_ER2xxx.Beckhoff_ER2xxxEK1122.A_0013_ER2038_0001_0018.WcState.WcState <-> WcState/WcState
//     PlcTask Inputs/GVL_iXlinker.EtherCAT_Master_ERxxxx.Beckhoff_ER2xxx.Beckhoff_ER2xxxEK1122.A_0013_ER2038_0001_0018.WcState.InputToggle <-> WcState/InputToggle
//     PlcTask Inputs/GVL_iXlinker.EtherCAT_Master_ERxxxx.Beckhoff_ER2xxx.Beckhoff_ER2xxxEK1122.A_0013_ER2038_0001_0018.InfoData.State <-> InfoData/State
//   PLC/PLC Instance <-> EtherCAT Master ERxxxx/Beckhoff ER2xxx/Beckhoff ER2xxxEK1122/A_0014(ER2038-0002-0017)
//     PlcTask Inputs/GVL_iXlinker.EtherCAT_Master_ERxxxx.Beckhoff_ER2xxx.Beckhoff_ER2xxxEK1122.A_0014_ER2038_0002_0017.Diag_Channel_1.Input <-> Diag Channel 1/Input
//     PlcTask Inputs/GVL_iXlinker.EtherCAT_Master_ERxxxx.Beckhoff_ER2xxx.Beckhoff_ER2xxxEK1122.A_0014_ER2038_0002_0017.Diag_Channel_2.Input <-> Diag Channel 2/Input
//     PlcTask Inputs/GVL_iXlinker.EtherCAT_Master_ERxxxx.Beckhoff_ER2xxx.Beckhoff_ER2xxxEK1122.A_0014_ER2038_0002_0017.Diag_Channel_3.Input <-> Diag Channel 3/Input
//     PlcTask Inputs/GVL_iXlinker.EtherCAT_Master_ERxxxx.Beckhoff_ER2xxx.Beckhoff_ER2xxxEK1122.A_0014_ER2038_0002_0017.Diag_Channel_4.Input <-> Diag Channel 4/Input
//     PlcTask Inputs/GVL_iXlinker.EtherCAT_Master_ERxxxx.Beckhoff_ER2xxx.Beckhoff_ER2xxxEK1122.A_0014_ER2038_0002_0017.Diag_Channel_5.Input <-> Diag Channel 5/Input
//     PlcTask Inputs/GVL_iXlinker.EtherCAT_Master_ERxxxx.Beckhoff_ER2xxx.Beckhoff_ER2xxxEK1122.A_0014_ER2038_0002_0017.Diag_Channel_6.Input <-> Diag Channel 6/Input
//     PlcTask Inputs/GVL_iXlinker.EtherCAT_Master_ERxxxx.Beckhoff_ER2xxx.Beckhoff_ER2xxxEK1122.A_0014_ER2038_0002_0017.Diag_Channel_7.Input <-> Diag Channel 7/Input
//     PlcTask Inputs/GVL_iXlinker.EtherCAT_Master_ERxxxx.Beckhoff_ER2xxx.Beckhoff_ER2xxxEK1122.A_0014_ER2038_0002_0017.Diag_Channel_8.Input <-> Diag Channel 8/Input
//     PlcTask Outputs/GVL_iXlinker.EtherCAT_Master_ERxxxx.Beckhoff_ER2xxx.Beckhoff_ER2xxxEK1122.A_0014_ER2038_0002_0017.Channel_1.Output <-> Channel 1/Output
//     PlcTask Outputs/GVL_iXlinker.EtherCAT_Master_ERxxxx.Beckhoff_ER2xxx.Beckhoff_ER2xxxEK1122.A_0014_ER2038_0002_0017.Channel_2.Output <-> Channel 2/Output
//     PlcTask Outputs/GVL_iXlinker.EtherCAT_Master_ERxxxx.Beckhoff_ER2xxx.Beckhoff_ER2xxxEK1122.A_0014_ER2038_0002_0017.Channel_3.Output <-> Channel 3/Output
//     PlcTask Outputs/GVL_iXlinker.EtherCAT_Master_ERxxxx.Beckhoff_ER2xxx.Beckhoff_ER2xxxEK1122.A_0014_ER2038_0002_0017.Channel_4.Output <-> Channel 4/Output
//     PlcTask Outputs/GVL_iXlinker.EtherCAT_Master_ERxxxx.Beckhoff_ER2xxx.Beckhoff_ER2xxxEK1122.A_0014_ER2038_0002_0017.Channel_5.Output <-> Channel 5/Output
//     PlcTask Outputs/GVL_iXlinker.EtherCAT_Master_ERxxxx.Beckhoff_ER2xxx.Beckhoff_ER2xxxEK1122.A_0014_ER2038_0002_0017.Channel_6.Output <-> Channel 6/Output
//     PlcTask Outputs/GVL_iXlinker.EtherCAT_Master_ERxxxx.Beckhoff_ER2xxx.Beckhoff_ER2xxxEK1122.A_0014_ER2038_0002_0017.Channel_7.Output <-> Channel 7/Output
//     PlcTask Outputs/GVL_iXlinker.EtherCAT_Master_ERxxxx.Beckhoff_ER2xxx.Beckhoff_ER2xxxEK1122.A_0014_ER2038_0002_0017.Channel_8.Output <-> Channel 8/Output
//     PlcTask Inputs/GVL_iXlinker.EtherCAT_Master_ERxxxx.Beckhoff_ER2xxx.Beckhoff_ER2xxxEK1122.A_0014_ER2038_0002_0017.WcState.WcState <-> WcState/WcState
//     PlcTask Inputs/GVL_iXlinker.EtherCAT_Master_ERxxxx.Beckhoff_ER2xxx.Beckhoff_ER2xxxEK1122.A_0014_ER2038_0002_0017.WcState.InputToggle <-> WcState/InputToggle
//     PlcTask Inputs/GVL_iXlinker.EtherCAT_Master_ERxxxx.Beckhoff_ER2xxx.Beckhoff_ER2xxxEK1122.A_0014_ER2038_0002_0017.InfoData.State <-> InfoData/State
//   PLC/PLC Instance <-> EtherCAT Master ERxxxx/Beckhoff ER2xxx/Beckhoff ER2xxxEK1122/A_0015(ER2038-0002-0018)
//     PlcTask Inputs/GVL_iXlinker.EtherCAT_Master_ERxxxx.Beckhoff_ER2xxx.Beckhoff_ER2xxxEK1122.A_0015_ER2038_0002_0018.Diag_Channel_1.Input <-> Diag Channel 1/Input
//     PlcTask Inputs/GVL_iXlinker.EtherCAT_Master_ERxxxx.Beckhoff_ER2xxx.Beckhoff_ER2xxxEK1122.A_0015_ER2038_0002_0018.Diag_Channel_2.Input <-> Diag Channel 2/Input
//     PlcTask Inputs/GVL_iXlinker.EtherCAT_Master_ERxxxx.Beckhoff_ER2xxx.Beckhoff_ER2xxxEK1122.A_0015_ER2038_0002_0018.Diag_Channel_3.Input <-> Diag Channel 3/Input
